    CONST robtarget T4037:=[[56.500013,31.797210,37.750261],[1.000000,0.000000,0.000000,0.000000],[0,0,-1,0],[9E+09,9E+09,9E+09,9E+09,9E+09,9E+09]];
    CONST robtarget T4038:=[[55.000007,31.515698,37.750261],[1.000000,0.000000,0.000000,0.000000],[0,0,-1,0],[9E+09,9E+09,9E+09,9E+09,9E+09,9E+09]];
    CONST robtarget T4039:=[[55.000007,58.695406,37.750261],[1.000000,0.000000,0.000000,0.000000],[0,0,-1,0],[9E+09,9E+09,9E+09,9E+09,9E+09,9E+09]];
    CONST robtarget T4040:=[[53.500001,58.570181,37.750261],[1.000000,0.000000,0.000000,0.000000],[0,0,-1,0],[9E+09,9E+09,9E+09,9E+09,9E+09,9E+09]];
    CONST robtarget T4041:=[[53.500001,31.797216,37.750261],[1.000000,0.000000,0.000000,0.000000],[0,0,-1,0],[9E+09,9E+09,9E+09,9E+09,9E+09,9E+09]];
    CONST robtarget T4042:=[[51.999995,32.435962,37.750261],[1.000000,0.000000,0.000000,0.000000],[0,0,-1,0],[9E+09,9E+09,9E+09,9E+09,9E+09,9E+09]];
    CONST robtarget T4043:=[[51.999995,58.394476,37.750261],[1.000000,0.000000,0.000000,0.000000],[0,0,-1,0],[9E+09,9E+09,9E+09,9E+09,9E+09,9E+09]];
    CONST robtarget T4044:=[[50.499989,57.901720,37.750261],[1.000000,0.000000,0.000000,0.000000],[0,0,-1,0],[9E+09,9E+09,9E+09,9E+09,9E+09,9E+09]];
    CONST robtarget T4045:=[[50.499989,33.195292,37.750261],[1.000000,0.000000,0.000000,0.000000],[0,0,-1,0],[9E+09,9E+09,9E+09,9E+09,9E+09,9E+09]];
    CONST robtarget T4046:=[[48.999983,34.510328,37.750261],[1.000000,0.000000,0.000000,0.000000],[0,0,-1,0],[9E+09,9E+09,9E+09,9E+09,9E+09,9E+09]];
    CONST robtarget T4047:=[[48.999983,57.171733,37.750261],[1.000000,0.000000,0.000000,0.000000],[0,0,-1,0],[9E+09,9E+09,9E+09,9E+09,9E+09,9E+09]];
    CONST robtarget T4048:=[[47.499977,56.303173,37.750261],[1.000000,0.000000,0.000000,0.000000],[0,0,-1,0],[9E+09,9E+09,9E+09,9E+09,9E+09,9E+09]];
    CONST robtarget T4049:=[[47.499977,37.856224,37.750261],[1.000000,0.000000,0.000000,0.000000],[0,0,-1,0],[9E+09,9E+09,9E+09,9E+09,9E+09,9E+09]];
    CONST robtarget T4050:=[[45.999971,39.948571,37.750261],[1.000000,0.000000,0.000000,0.000000],[0,0,-1,0],[9E+09,9E+09,9E+09,9E+09,9E+09,9E+09]];
    CONST robtarget T4051:=[[45.999971,54.916021,37.750261],[1.000000,0.000000,0.000000,0.000000],[0,0,-1,0],[9E+09,9E+09,9E+09,9E+09,9E+09,9E+09]];
    CONST robtarget T4052:=[[44.499965,53.011141,37.750261],[1.000000,0.000000,0.000000,0.000000],[0,0,-1,0],[9E+09,9E+09,9E+09,9E+09,9E+09,9E+09]];
    CONST robtarget T4053:=[[44.499965,42.078797,37.750261],[1.000000,0.000000,0.000000,0.000000],[0,0,-1,0],[9E+09,9E+09,9E+09,9E+09,9E+09,9E+09]];
    CONST robtarget T4054:=[[42.999959,44.372557,37.750261],[1.000000,0.000000,0.000000,0.000000],[0,0,-1,0],[9E+09,9E+09,9E+09,9E+09,9E+09,9E+09]];
    CONST robtarget T4055:=[[42.999959,50.112291,37.750261],[1.000000,0.000000,0.000000,0.000000],[0,0,-1,0],[9E+09,9E+09,9E+09,9E+09,9E+09,9E+09]];
    CONST robtarget T4056:=[[42.999959,44.212149,38.250271],[1.000000,0.000000,0.000000,0.000000],[0,0,-1,0],[9E+09,9E+09,9E+09,9E+09,9E+09,9E+09]];
    CONST robtarget T4057:=[[42.999959,50.185983,38.250271],[1.000000,0.000000,0.000000,0.000000],[0,0,-1,0],[9E+09,9E+09,9E+09,9E+09,9E+09,9E+09]];
    CONST robtarget T4058:=[[42.999959,44.212149,38.250271],[1.000000,0.000000,0.000000,0.000000],[0,0,-1,0],[9E+09,9E+09,9E+09,9E+09,9E+09,9E+09]];
    CONST robtarget T4059:=[[42.999959,50.185983,38.250271],[1.000000,0.000000,0.000000,0.000000],[0,0,-1,0],[9E+09,9E+09,9E+09,9E+09,9E+09,9E+09]];
    CONST robtarget T4060:=[[44.499965,53.123117,38.250271],[1.000000,0.000000,0.000000,0.000000],[0,0,-1,0],[9E+09,9E+09,9E+09,9E+09,9E+09,9E+09]];
    CONST robtarget T4061:=[[44.499965,42.207669,38.250271],[1.000000,0.000000,0.000000,0.000000],[0,0,-1,0],[9E+09,9E+09,9E+09,9E+09,9E+09,9E+09]];
    CONST robtarget T4062:=[[45.999971,40.057127,38.250271],[1.000000,0.000000,0.000000,0.000000],[0,0,-1,0],[9E+09,9E+09,9E+09,9E+09,9E+09,9E+09]];
    CONST robtarget T4063:=[[45.999971,55.075491,38.250271],[1.000000,0.000000,0.000000,0.000000],[0,0,-1,0],[9E+09,9E+09,9E+09,9E+09,9E+09,9E+09]];
    CONST robtarget T4064:=[[47.499977,56.371057,38.250271],[1.000000,0.000000,0.000000,0.000000],[0,0,-1,0],[9E+09,9E+09,9E+09,9E+09,9E+09,9E+09]];
    CONST robtarget T4065:=[[47.499977,38.617217,38.250271],[1.000000,0.000000,0.000000,0.000000],[0,0,-1,0],[9E+09,9E+09,9E+09,9E+09,9E+09,9E+09]];
    CONST robtarget T4066:=[[48.999983,35.664766,38.250271],[1.000000,0.000000,0.000000,0.000000],[0,0,-1,0],[9E+09,9E+09,9E+09,9E+09,9E+09,9E+09]];
    CONST robtarget T4067:=[[48.999983,57.294926,38.250271],[1.000000,0.000000,0.000000,0.000000],[0,0,-1,0],[9E+09,9E+09,9E+09,9E+09,9E+09,9E+09]];
    CONST robtarget T4068:=[[50.499989,58.002093,38.250271],[1.000000,0.000000,0.000000,0.000000],[0,0,-1,0],[9E+09,9E+09,9E+09,9E+09,9E+09,9E+09]];
    CONST robtarget T4069:=[[50.499989,32.700822,38.250271],[1.000000,0.000000,0.000000,0.000000],[0,0,-1,0],[9E+09,9E+09,9E+09,9E+09,9E+09,9E+09]];
    CONST robtarget T4070:=[[51.999995,32.054897,38.250271],[1.000000,0.000000,0.000000,0.000000],[0,0,-1,0],[9E+09,9E+09,9E+09,9E+09,9E+09,9E+09]];
    CONST robtarget T4071:=[[51.999995,58.459231,38.250271],[1.000000,0.000000,0.000000,0.000000],[0,0,-1,0],[9E+09,9E+09,9E+09,9E+09,9E+09,9E+09]];
    CONST robtarget T4072:=[[53.500001,58.647265,38.250271],[1.000000,0.000000,0.000000,0.000000],[0,0,-1,0],[9E+09,9E+09,9E+09,9E+09,9E+09,9E+09]];
    CONST robtarget T4073:=[[53.500001,31.359567,38.250271],[1.000000,0.000000,0.000000,0.000000],[0,0,-1,0],[9E+09,9E+09,9E+09,9E+09,9E+09,9E+09]];
    CONST robtarget T4074:=[[55.000007,31.064300,38.250271],[1.000000,0.000000,0.000000,0.000000],[0,0,-1,0],[9E+09,9E+09,9E+09,9E+09,9E+09,9E+09]];
    CONST robtarget T4075:=[[55.000007,58.772490,38.250271],[1.000000,0.000000,0.000000,0.000000],[0,0,-1,0],[9E+09,9E+09,9E+09,9E+09,9E+09,9E+09]];
    CONST robtarget T4076:=[[56.500013,58.647265,38.250271],[1.000000,0.000000,0.000000,0.000000],[0,0,-1,0],[9E+09,9E+09,9E+09,9E+09,9E+09,9E+09]];
    CONST robtarget T4077:=[[56.500013,31.359567,38.250271],[1.000000,0.000000,0.000000,0.000000],[0,0,-1,0],[9E+09,9E+09,9E+09,9E+09,9E+09,9E+09]];
    CONST robtarget T4078:=[[58.000019,32.054894,38.250271],[1.000000,0.000000,0.000000,0.000000],[0,0,-1,0],[9E+09,9E+09,9E+09,9E+09,9E+09,9E+09]];
    CONST robtarget T4079:=[[58.000019,58.459229,38.250271],[1.000000,0.000000,0.000000,0.000000],[0,0,-1,0],[9E+09,9E+09,9E+09,9E+09,9E+09,9E+09]];
    CONST robtarget T4080:=[[59.500025,58.002093,38.250271],[1.000000,0.000000,0.000000,0.000000],[0,0,-1,0],[9E+09,9E+09,9E+09,9E+09,9E+09,9E+09]];
    CONST robtarget T4081:=[[59.500025,32.700830,38.250271],[1.000000,0.000000,0.000000,0.000000],[0,0,-1,0],[9E+09,9E+09,9E+09,9E+09,9E+09,9E+09]];
    CONST robtarget T4082:=[[61.000031,35.664766,38.250271],[1.000000,0.000000,0.000000,0.000000],[0,0,-1,0],[9E+09,9E+09,9E+09,9E+09,9E+09,9E+09]];
    CONST robtarget T4083:=[[61.000031,57.294925,38.250271],[1.000000,0.000000,0.000000,0.000000],[0,0,-1,0],[9E+09,9E+09,9E+09,9E+09,9E+09,9E+09]];
    CONST robtarget T4084:=[[62.500037,56.371056,38.250271],[1.000000,0.000000,0.000000,0.000000],[0,0,-1,0],[9E+09,9E+09,9E+09,9E+09,9E+09,9E+09]];
    CONST robtarget T4085:=[[62.500037,38.617217,38.250271],[1.000000,0.000000,0.000000,0.000000],[0,0,-1,0],[9E+09,9E+09,9E+09,9E+09,9E+09,9E+09]];
    CONST robtarget T4086:=[[64.000043,40.057127,38.250271],[1.000000,0.000000,0.000000,0.000000],[0,0,-1,0],[9E+09,9E+09,9E+09,9E+09,9E+09,9E+09]];
    CONST robtarget T4087:=[[64.000043,55.075491,38.250271],[1.000000,0.000000,0.000000,0.000000],[0,0,-1,0],[9E+09,9E+09,9E+09,9E+09,9E+09,9E+09]];
    CONST robtarget T4088:=[[65.500049,53.123116,38.250271],[1.000000,0.000000,0.000000,0.000000],[0,0,-1,0],[9E+09,9E+09,9E+09,9E+09,9E+09,9E+09]];
    CONST robtarget T4089:=[[65.500049,42.207669,38.250271],[1.000000,0.000000,0.000000,0.000000],[0,0,-1,0],[9E+09,9E+09,9E+09,9E+09,9E+09,9E+09]];
    CONST robtarget T4090:=[[67.000055,44.212149,38.250271],[1.000000,0.000000,0.000000,0.000000],[0,0,-1,0],[9E+09,9E+09,9E+09,9E+09,9E+09,9E+09]];
    CONST robtarget T4091:=[[67.000055,50.185984,38.250271],[1.000000,0.000000,0.000000,0.000000],[0,0,-1,0],[9E+09,9E+09,9E+09,9E+09,9E+09,9E+09]];
    CONST robtarget T4092:=[[67.000055,44.131949,38.750281],[1.000000,0.000000,0.000000,0.000000],[0,0,-1,0],[9E+09,9E+09,9E+09,9E+09,9E+09,9E+09]];
    CONST robtarget T4093:=[[67.000055,50.259676,38.750281],[1.000000,0.000000,0.000000,0.000000],[0,0,-1,0],[9E+09,9E+09,9E+09,9E+09,9E+09,9E+09]];
    CONST robtarget T4094:=[[67.000055,44.131949,38.750281],[1.000000,0.000000,0.000000,0.000000],[0,0,-1,0],[9E+09,9E+09,9E+09,9E+09,9E+09,9E+09]];
    CONST robtarget T4095:=[[67.000055,50.259676,38.750281],[1.000000,0.000000,0.000000,0.000000],[0,0,-1,0],[9E+09,9E+09,9E+09,9E+09,9E+09,9E+09]];
    CONST robtarget T4096:=[[65.500049,53.235088,38.750281],[1.000000,0.000000,0.000000,0.000000],[0,0,-1,0],[9E+09,9E+09,9E+09,9E+09,9E+09,9E+09]];
    CONST robtarget T4097:=[[65.500049,42.336541,38.750281],[1.000000,0.000000,0.000000,0.000000],[0,0,-1,0],[9E+09,9E+09,9E+09,9E+09,9E+09,9E+09]];
    CONST robtarget T4098:=[[64.000043,40.167265,38.750281],[1.000000,0.000000,0.000000,0.000000],[0,0,-1,0],[9E+09,9E+09,9E+09,9E+09,9E+09,9E+09]];
    CONST robtarget T4099:=[[64.000043,55.123261,38.750281],[1.000000,0.000000,0.000000,0.000000],[0,0,-1,0],[9E+09,9E+09,9E+09,9E+09,9E+09,9E+09]];
    CONST robtarget T4100:=[[62.500037,56.438940,38.750281],[1.000000,0.000000,0.000000,0.000000],[0,0,-1,0],[9E+09,9E+09,9E+09,9E+09,9E+09,9E+09]];
    CONST robtarget T4101:=[[62.500037,38.816896,38.750281],[1.000000,0.000000,0.000000,0.000000],[0,0,-1,0],[9E+09,9E+09,9E+09,9E+09,9E+09,9E+09]];
    CONST robtarget T4102:=[[61.000031,36.698545,38.750281],[1.000000,0.000000,0.000000,0.000000],[0,0,-1,0],[9E+09,9E+09,9E+09,9E+09,9E+09,9E+09]];
    CONST robtarget T4103:=[[61.000031,57.398916,38.750281],[1.000000,0.000000,0.000000,0.000000],[0,0,-1,0],[9E+09,9E+09,9E+09,9E+09,9E+09,9E+09]];
    CONST robtarget T4104:=[[59.500025,58.045436,38.750281],[1.000000,0.000000,0.000000,0.000000],[0,0,-1,0],[9E+09,9E+09,9E+09,9E+09,9E+09,9E+09]];
    CONST robtarget T4105:=[[59.500025,32.999058,38.750281],[1.000000,0.000000,0.000000,0.000000],[0,0,-1,0],[9E+09,9E+09,9E+09,9E+09,9E+09,9E+09]];
    CONST robtarget T4106:=[[58.000019,31.695724,38.750281],[1.000000,0.000000,0.000000,0.000000],[0,0,-1,0],[9E+09,9E+09,9E+09,9E+09,9E+09,9E+09]];
    CONST robtarget T4107:=[[58.000019,58.532197,38.750281],[1.000000,0.000000,0.000000,0.000000],[0,0,-1,0],[9E+09,9E+09,9E+09,9E+09,9E+09,9E+09]];
    CONST robtarget T4108:=[[56.500013,58.721504,38.750281],[1.000000,0.000000,0.000000,0.000000],[0,0,-1,0],[9E+09,9E+09,9E+09,9E+09,9E+09,9E+09]];
    CONST robtarget T4109:=[[56.500013,30.999539,38.750281],[1.000000,0.000000,0.000000,0.000000],[0,0,-1,0],[9E+09,9E+09,9E+09,9E+09,9E+09,9E+09]];
    CONST robtarget T4110:=[[55.000007,30.672510,38.750281],[1.000000,0.000000,0.000000,0.000000],[0,0,-1,0],[9E+09,9E+09,9E+09,9E+09,9E+09,9E+09]];
    CONST robtarget T4111:=[[55.000007,58.849574,38.750281],[1.000000,0.000000,0.000000,0.000000],[0,0,-1,0],[9E+09,9E+09,9E+09,9E+09,9E+09,9E+09]];
    CONST robtarget T4112:=[[53.500001,58.721507,38.750281],[1.000000,0.000000,0.000000,0.000000],[0,0,-1,0],[9E+09,9E+09,9E+09,9E+09,9E+09,9E+09]];
    CONST robtarget T4113:=[[53.500001,30.999539,38.750281],[1.000000,0.000000,0.000000,0.000000],[0,0,-1,0],[9E+09,9E+09,9E+09,9E+09,9E+09,9E+09]];
    CONST robtarget T4114:=[[51.999995,31.695723,38.750281],[1.000000,0.000000,0.000000,0.000000],[0,0,-1,0],[9E+09,9E+09,9E+09,9E+09,9E+09,9E+09]];
    CONST robtarget T4115:=[[51.999995,58.532203,38.750281],[1.000000,0.000000,0.000000,0.000000],[0,0,-1,0],[9E+09,9E+09,9E+09,9E+09,9E+09,9E+09]];
    CONST robtarget T4116:=[[50.499989,58.045436,38.750281],[1.000000,0.000000,0.000000,0.000000],[0,0,-1,0],[9E+09,9E+09,9E+09,9E+09,9E+09,9E+09]];
    CONST robtarget T4117:=[[50.499989,32.999059,38.750281],[1.000000,0.000000,0.000000,0.000000],[0,0,-1,0],[9E+09,9E+09,9E+09,9E+09,9E+09,9E+09]];
    CONST robtarget T4118:=[[48.999983,36.698544,38.750281],[1.000000,0.000000,0.000000,0.000000],[0,0,-1,0],[9E+09,9E+09,9E+09,9E+09,9E+09,9E+09]];
    CONST robtarget T4119:=[[48.999983,57.398916,38.750281],[1.000000,0.000000,0.000000,0.000000],[0,0,-1,0],[9E+09,9E+09,9E+09,9E+09,9E+09,9E+09]];
    CONST robtarget T4120:=[[47.499977,56.438941,38.750281],[1.000000,0.000000,0.000000,0.000000],[0,0,-1,0],[9E+09,9E+09,9E+09,9E+09,9E+09,9E+09]];
    CONST robtarget T4121:=[[47.499977,38.816896,38.750281],[1.000000,0.000000,0.000000,0.000000],[0,0,-1,0],[9E+09,9E+09,9E+09,9E+09,9E+09,9E+09]];
    CONST robtarget T4122:=[[45.999971,40.167264,38.750281],[1.000000,0.000000,0.000000,0.000000],[0,0,-1,0],[9E+09,9E+09,9E+09,9E+09,9E+09,9E+09]];
    CONST robtarget T4123:=[[45.999971,55.123261,38.750281],[1.000000,0.000000,0.000000,0.000000],[0,0,-1,0],[9E+09,9E+09,9E+09,9E+09,9E+09,9E+09]];
    CONST robtarget T4124:=[[44.499965,53.235093,38.750281],[1.000000,0.000000,0.000000,0.000000],[0,0,-1,0],[9E+09,9E+09,9E+09,9E+09,9E+09,9E+09]];
    CONST robtarget T4125:=[[44.499965,42.336540,38.750281],[1.000000,0.000000,0.000000,0.000000],[0,0,-1,0],[9E+09,9E+09,9E+09,9E+09,9E+09,9E+09]];
    CONST robtarget T4126:=[[42.999959,44.131948,38.750281],[1.000000,0.000000,0.000000,0.000000],[0,0,-1,0],[9E+09,9E+09,9E+09,9E+09,9E+09,9E+09]];
    CONST robtarget T4127:=[[42.999959,50.259676,38.750281],[1.000000,0.000000,0.000000,0.000000],[0,0,-1,0],[9E+09,9E+09,9E+09,9E+09,9E+09,9E+09]];
    CONST robtarget T4128:=[[42.999959,44.054116,39.250291],[1.000000,0.000000,0.000000,0.000000],[0,0,-1,0],[9E+09,9E+09,9E+09,9E+09,9E+09,9E+09]];
    CONST robtarget T4129:=[[42.999959,50.376289,39.250291],[1.000000,0.000000,0.000000,0.000000],[0,0,-1,0],[9E+09,9E+09,9E+09,9E+09,9E+09,9E+09]];
    CONST robtarget T4130:=[[42.999959,44.054116,39.250291],[1.000000,0.000000,0.000000,0.000000],[0,0,-1,0],[9E+09,9E+09,9E+09,9E+09,9E+09,9E+09]];
    CONST robtarget T4131:=[[42.999959,50.376289,39.250291],[1.000000,0.000000,0.000000,0.000000],[0,0,-1,0],[9E+09,9E+09,9E+09,9E+09,9E+09,9E+09]];
    CONST robtarget T4132:=[[44.499965,53.135053,39.250291],[1.000000,0.000000,0.000000,0.000000],[0,0,-1,0],[9E+09,9E+09,9E+09,9E+09,9E+09,9E+09]];
    CONST robtarget T4133:=[[44.499965,42.332431,39.250291],[1.000000,0.000000,0.000000,0.000000],[0,0,-1,0],[9E+09,9E+09,9E+09,9E+09,9E+09,9E+09]];
    CONST robtarget T4134:=[[45.999971,40.374790,39.250291],[1.000000,0.000000,0.000000,0.000000],[0,0,-1,0],[9E+09,9E+09,9E+09,9E+09,9E+09,9E+09]];
    CONST robtarget T4135:=[[45.999971,55.113414,39.250291],[1.000000,0.000000,0.000000,0.000000],[0,0,-1,0],[9E+09,9E+09,9E+09,9E+09,9E+09,9E+09]];
    CONST robtarget T4136:=[[47.499977,56.506825,39.250291],[1.000000,0.000000,0.000000,0.000000],[0,0,-1,0],[9E+09,9E+09,9E+09,9E+09,9E+09,9E+09]];
    CONST robtarget T4137:=[[47.499977,38.996522,39.250291],[1.000000,0.000000,0.000000,0.000000],[0,0,-1,0],[9E+09,9E+09,9E+09,9E+09,9E+09,9E+09]];
    CONST robtarget T4138:=[[48.999983,37.580618,39.250291],[1.000000,0.000000,0.000000,0.000000],[0,0,-1,0],[9E+09,9E+09,9E+09,9E+09,9E+09,9E+09]];
    CONST robtarget T4139:=[[48.999983,57.420832,39.250291],[1.000000,0.000000,0.000000,0.000000],[0,0,-1,0],[9E+09,9E+09,9E+09,9E+09,9E+09,9E+09]];
    CONST robtarget T4140:=[[50.499989,58.088778,39.250291],[1.000000,0.000000,0.000000,0.000000],[0,0,-1,0],[9E+09,9E+09,9E+09,9E+09,9E+09,9E+09]];
    CONST robtarget T4141:=[[50.499989,34.138448,39.250291],[1.000000,0.000000,0.000000,0.000000],[0,0,-1,0],[9E+09,9E+09,9E+09,9E+09,9E+09,9E+09]];
    CONST robtarget T4142:=[[51.999995,31.384926,39.250291],[1.000000,0.000000,0.000000,0.000000],[0,0,-1,0],[9E+09,9E+09,9E+09,9E+09,9E+09,9E+09]];
    CONST robtarget T4143:=[[51.999995,58.605174,39.250291],[1.000000,0.000000,0.000000,0.000000],[0,0,-1,0],[9E+09,9E+09,9E+09,9E+09,9E+09,9E+09]];
    CONST robtarget T4144:=[[53.500001,58.780455,39.250291],[1.000000,0.000000,0.000000,0.000000],[0,0,-1,0],[9E+09,9E+09,9E+09,9E+09,9E+09,9E+09]];
    CONST robtarget T4145:=[[53.500001,30.721918,39.250291],[1.000000,0.000000,0.000000,0.000000],[0,0,-1,0],[9E+09,9E+09,9E+09,9E+09,9E+09,9E+09]];
    CONST robtarget T4146:=[[55.000007,30.347257,39.250291],[1.000000,0.000000,0.000000,0.000000],[0,0,-1,0],[9E+09,9E+09,9E+09,9E+09,9E+09,9E+09]];
    CONST robtarget T4147:=[[55.000007,58.890261,39.250291],[1.000000,0.000000,0.000000,0.000000],[0,0,-1,0],[9E+09,9E+09,9E+09,9E+09,9E+09,9E+09]];
    CONST robtarget T4148:=[[56.500013,58.780450,39.250291],[1.000000,0.000000,0.000000,0.000000],[0,0,-1,0],[9E+09,9E+09,9E+09,9E+09,9E+09,9E+09]];
    CONST robtarget T4149:=[[56.500013,30.721922,39.250291],[1.000000,0.000000,0.000000,0.000000],[0,0,-1,0],[9E+09,9E+09,9E+09,9E+09,9E+09,9E+09]];
    CONST robtarget T4150:=[[58.000019,31.384926,39.250291],[1.000000,0.000000,0.000000,0.000000],[0,0,-1,0],[9E+09,9E+09,9E+09,9E+09,9E+09,9E+09]];
    CONST robtarget T4151:=[[58.000019,58.605166,39.250291],[1.000000,0.000000,0.000000,0.000000],[0,0,-1,0],[9E+09,9E+09,9E+09,9E+09,9E+09,9E+09]];
    CONST robtarget T4152:=[[59.500025,58.088778,39.250291],[1.000000,0.000000,0.000000,0.000000],[0,0,-1,0],[9E+09,9E+09,9E+09,9E+09,9E+09,9E+09]];
    CONST robtarget T4153:=[[59.500025,34.138448,39.250291],[1.000000,0.000000,0.000000,0.000000],[0,0,-1,0],[9E+09,9E+09,9E+09,9E+09,9E+09,9E+09]];
    CONST robtarget T4154:=[[61.000031,37.580618,39.250291],[1.000000,0.000000,0.000000,0.000000],[0,0,-1,0],[9E+09,9E+09,9E+09,9E+09,9E+09,9E+09]];
    CONST robtarget T4155:=[[61.000031,57.420832,39.250291],[1.000000,0.000000,0.000000,0.000000],[0,0,-1,0],[9E+09,9E+09,9E+09,9E+09,9E+09,9E+09]];
    CONST robtarget T4156:=[[62.500037,56.506824,39.250291],[1.000000,0.000000,0.000000,0.000000],[0,0,-1,0],[9E+09,9E+09,9E+09,9E+09,9E+09,9E+09]];
    CONST robtarget T4157:=[[62.500037,38.996523,39.250291],[1.000000,0.000000,0.000000,0.000000],[0,0,-1,0],[9E+09,9E+09,9E+09,9E+09,9E+09,9E+09]];
    CONST robtarget T4158:=[[64.000043,40.374792,39.250291],[1.000000,0.000000,0.000000,0.000000],[0,0,-1,0],[9E+09,9E+09,9E+09,9E+09,9E+09,9E+09]];
    CONST robtarget T4159:=[[64.000043,55.113414,39.250291],[1.000000,0.000000,0.000000,0.000000],[0,0,-1,0],[9E+09,9E+09,9E+09,9E+09,9E+09,9E+09]];
    CONST robtarget T4160:=[[65.500049,53.135049,39.250291],[1.000000,0.000000,0.000000,0.000000],[0,0,-1,0],[9E+09,9E+09,9E+09,9E+09,9E+09,9E+09]];
    CONST robtarget T4161:=[[65.500049,42.332431,39.250291],[1.000000,0.000000,0.000000,0.000000],[0,0,-1,0],[9E+09,9E+09,9E+09,9E+09,9E+09,9E+09]];
    CONST robtarget T4162:=[[67.000055,44.054117,39.250291],[1.000000,0.000000,0.000000,0.000000],[0,0,-1,0],[9E+09,9E+09,9E+09,9E+09,9E+09,9E+09]];
    CONST robtarget T4163:=[[67.000055,50.376286,39.250291],[1.000000,0.000000,0.000000,0.000000],[0,0,-1,0],[9E+09,9E+09,9E+09,9E+09,9E+09,9E+09]];
    CONST robtarget T4164:=[[67.000055,44.072887,39.750301],[1.000000,0.000000,0.000000,0.000000],[0,0,-1,0],[9E+09,9E+09,9E+09,9E+09,9E+09,9E+09]];
    CONST robtarget T4165:=[[67.000055,50.303617,39.750301],[1.000000,0.000000,0.000000,0.000000],[0,0,-1,0],[9E+09,9E+09,9E+09,9E+09,9E+09,9E+09]];
    CONST robtarget T4166:=[[67.000055,44.072887,39.750301],[1.000000,0.000000,0.000000,0.000000],[0,0,-1,0],[9E+09,9E+09,9E+09,9E+09,9E+09,9E+09]];
    CONST robtarget T4167:=[[67.000055,50.303617,39.750301],[1.000000,0.000000,0.000000,0.000000],[0,0,-1,0],[9E+09,9E+09,9E+09,9E+09,9E+09,9E+09]];
    CONST robtarget T4168:=[[65.500049,52.995505,39.750301],[1.000000,0.000000,0.000000,0.000000],[0,0,-1,0],[9E+09,9E+09,9E+09,9E+09,9E+09,9E+09]];
    CONST robtarget T4169:=[[65.500049,42.422914,39.750301],[1.000000,0.000000,0.000000,0.000000],[0,0,-1,0],[9E+09,9E+09,9E+09,9E+09,9E+09,9E+09]];
    CONST robtarget T4170:=[[64.000043,40.653208,39.750301],[1.000000,0.000000,0.000000,0.000000],[0,0,-1,0],[9E+09,9E+09,9E+09,9E+09,9E+09,9E+09]];
    CONST robtarget T4171:=[[64.000043,55.084923,39.750301],[1.000000,0.000000,0.000000,0.000000],[0,0,-1,0],[9E+09,9E+09,9E+09,9E+09,9E+09,9E+09]];
    CONST robtarget T4172:=[[62.500037,56.521256,39.750301],[1.000000,0.000000,0.000000,0.000000],[0,0,-1,0],[9E+09,9E+09,9E+09,9E+09,9E+09,9E+09]];
    CONST robtarget T4173:=[[62.500037,39.193232,39.750301],[1.000000,0.000000,0.000000,0.000000],[0,0,-1,0],[9E+09,9E+09,9E+09,9E+09,9E+09,9E+09]];
    CONST robtarget T4174:=[[61.000031,38.058259,39.750301],[1.000000,0.000000,0.000000,0.000000],[0,0,-1,0],[9E+09,9E+09,9E+09,9E+09,9E+09,9E+09]];
    CONST robtarget T4175:=[[61.000031,57.442748,39.750301],[1.000000,0.000000,0.000000,0.000000],[0,0,-1,0],[9E+09,9E+09,9E+09,9E+09,9E+09,9E+09]];
    CONST robtarget T4176:=[[59.500025,58.151010,39.750301],[1.000000,0.000000,0.000000,0.000000],[0,0,-1,0],[9E+09,9E+09,9E+09,9E+09,9E+09,9E+09]];
    CONST robtarget T4177:=[[59.500025,35.190368,39.750301],[1.000000,0.000000,0.000000,0.000000],[0,0,-1,0],[9E+09,9E+09,9E+09,9E+09,9E+09,9E+09]];
    CONST robtarget T4178:=[[58.000019,31.632069,39.750301],[1.000000,0.000000,0.000000,0.000000],[0,0,-1,0],[9E+09,9E+09,9E+09,9E+09,9E+09,9E+09]];
    CONST robtarget T4179:=[[58.000019,58.594733,39.750301],[1.000000,0.000000,0.000000,0.000000],[0,0,-1,0],[9E+09,9E+09,9E+09,9E+09,9E+09,9E+09]];
    CONST robtarget T4180:=[[56.500013,58.779478,39.750301],[1.000000,0.000000,0.000000,0.000000],[0,0,-1,0],[9E+09,9E+09,9E+09,9E+09,9E+09,9E+09]];
    CONST robtarget T4181:=[[56.500013,30.692136,39.750301],[1.000000,0.000000,0.000000,0.000000],[0,0,-1,0],[9E+09,9E+09,9E+09,9E+09,9E+09,9E+09]];
    CONST robtarget T4182:=[[55.000007,30.109747,39.750301],[1.000000,0.000000,0.000000,0.000000],[0,0,-1,0],[9E+09,9E+09,9E+09,9E+09,9E+09,9E+09]];
    CONST robtarget T4183:=[[55.000007,58.885895,39.750301],[1.000000,0.000000,0.000000,0.000000],[0,0,-1,0],[9E+09,9E+09,9E+09,9E+09,9E+09,9E+09]];
    CONST robtarget T4184:=[[53.500001,58.779480,39.750301],[1.000000,0.000000,0.000000,0.000000],[0,0,-1,0],[9E+09,9E+09,9E+09,9E+09,9E+09,9E+09]];
    CONST robtarget T4185:=[[53.500001,30.692135,39.750301],[1.000000,0.000000,0.000000,0.000000],[0,0,-1,0],[9E+09,9E+09,9E+09,9E+09,9E+09,9E+09]];
    CONST robtarget T4186:=[[51.999995,31.632069,39.750301],[1.000000,0.000000,0.000000,0.000000],[0,0,-1,0],[9E+09,9E+09,9E+09,9E+09,9E+09,9E+09]];
    CONST robtarget T4187:=[[51.999995,58.594739,39.750301],[1.000000,0.000000,0.000000,0.000000],[0,0,-1,0],[9E+09,9E+09,9E+09,9E+09,9E+09,9E+09]];
    CONST robtarget T4188:=[[50.499989,58.151012,39.750301],[1.000000,0.000000,0.000000,0.000000],[0,0,-1,0],[9E+09,9E+09,9E+09,9E+09,9E+09,9E+09]];
    CONST robtarget T4189:=[[50.499989,35.190377,39.750301],[1.000000,0.000000,0.000000,0.000000],[0,0,-1,0],[9E+09,9E+09,9E+09,9E+09,9E+09,9E+09]];
    CONST robtarget T4190:=[[48.999983,38.058258,39.750301],[1.000000,0.000000,0.000000,0.000000],[0,0,-1,0],[9E+09,9E+09,9E+09,9E+09,9E+09,9E+09]];
    CONST robtarget T4191:=[[48.999983,57.442748,39.750301],[1.000000,0.000000,0.000000,0.000000],[0,0,-1,0],[9E+09,9E+09,9E+09,9E+09,9E+09,9E+09]];
    CONST robtarget T4192:=[[47.499977,56.521257,39.750301],[1.000000,0.000000,0.000000,0.000000],[0,0,-1,0],[9E+09,9E+09,9E+09,9E+09,9E+09,9E+09]];
    CONST robtarget T4193:=[[47.499977,39.193232,39.750301],[1.000000,0.000000,0.000000,0.000000],[0,0,-1,0],[9E+09,9E+09,9E+09,9E+09,9E+09,9E+09]];
    CONST robtarget T4194:=[[45.999971,40.653206,39.750301],[1.000000,0.000000,0.000000,0.000000],[0,0,-1,0],[9E+09,9E+09,9E+09,9E+09,9E+09,9E+09]];
    CONST robtarget T4195:=[[45.999971,55.084923,39.750301],[1.000000,0.000000,0.000000,0.000000],[0,0,-1,0],[9E+09,9E+09,9E+09,9E+09,9E+09,9E+09]];
    CONST robtarget T4196:=[[44.499965,52.995507,39.750301],[1.000000,0.000000,0.000000,0.000000],[0,0,-1,0],[9E+09,9E+09,9E+09,9E+09,9E+09,9E+09]];
    CONST robtarget T4197:=[[44.499965,42.422914,39.750301],[1.000000,0.000000,0.000000,0.000000],[0,0,-1,0],[9E+09,9E+09,9E+09,9E+09,9E+09,9E+09]];
    CONST robtarget T4198:=[[42.999959,44.072887,39.750301],[1.000000,0.000000,0.000000,0.000000],[0,0,-1,0],[9E+09,9E+09,9E+09,9E+09,9E+09,9E+09]];
    CONST robtarget T4199:=[[42.999959,50.303618,39.750301],[1.000000,0.000000,0.000000,0.000000],[0,0,-1,0],[9E+09,9E+09,9E+09,9E+09,9E+09,9E+09]];
    CONST robtarget T4200:=[[42.999959,43.957416,40.250311],[1.000000,0.000000,0.000000,0.000000],[0,0,-1,0],[9E+09,9E+09,9E+09,9E+09,9E+09,9E+09]];
    CONST robtarget T4201:=[[42.999959,50.041103,40.250311],[1.000000,0.000000,0.000000,0.000000],[0,0,-1,0],[9E+09,9E+09,9E+09,9E+09,9E+09,9E+09]];
    CONST robtarget T4202:=[[42.999959,43.957416,40.250311],[1.000000,0.000000,0.000000,0.000000],[0,0,-1,0],[9E+09,9E+09,9E+09,9E+09,9E+09,9E+09]];
    CONST robtarget T4203:=[[42.999959,50.041103,40.250311],[1.000000,0.000000,0.000000,0.000000],[0,0,-1,0],[9E+09,9E+09,9E+09,9E+09,9E+09,9E+09]];
    CONST robtarget T4204:=[[44.499965,52.855961,40.250311],[1.000000,0.000000,0.000000,0.000000],[0,0,-1,0],[9E+09,9E+09,9E+09,9E+09,9E+09,9E+09]];
    CONST robtarget T4205:=[[44.499965,42.549901,40.250311],[1.000000,0.000000,0.000000,0.000000],[0,0,-1,0],[9E+09,9E+09,9E+09,9E+09,9E+09,9E+09]];
    CONST robtarget T4206:=[[45.999971,40.933620,40.250311],[1.000000,0.000000,0.000000,0.000000],[0,0,-1,0],[9E+09,9E+09,9E+09,9E+09,9E+09,9E+09]];
    CONST robtarget T4207:=[[45.999971,55.056432,40.250311],[1.000000,0.000000,0.000000,0.000000],[0,0,-1,0],[9E+09,9E+09,9E+09,9E+09,9E+09,9E+09]];
    CONST robtarget T4208:=[[47.499977,56.418593,40.250311],[1.000000,0.000000,0.000000,0.000000],[0,0,-1,0],[9E+09,9E+09,9E+09,9E+09,9E+09,9E+09]];
    CONST robtarget T4209:=[[47.499977,39.361755,40.250311],[1.000000,0.000000,0.000000,0.000000],[0,0,-1,0],[9E+09,9E+09,9E+09,9E+09,9E+09,9E+09]];
    CONST robtarget T4210:=[[48.999983,38.258018,40.250311],[1.000000,0.000000,0.000000,0.000000],[0,0,-1,0],[9E+09,9E+09,9E+09,9E+09,9E+09,9E+09]];
    CONST robtarget T4211:=[[48.999983,57.406745,40.250311],[1.000000,0.000000,0.000000,0.000000],[0,0,-1,0],[9E+09,9E+09,9E+09,9E+09,9E+09,9E+09]];
    CONST robtarget T4212:=[[50.499989,58.142889,40.250311],[1.000000,0.000000,0.000000,0.000000],[0,0,-1,0],[9E+09,9E+09,9E+09,9E+09,9E+09,9E+09]];
    CONST robtarget T4213:=[[50.499989,36.203320,40.250311],[1.000000,0.000000,0.000000,0.000000],[0,0,-1,0],[9E+09,9E+09,9E+09,9E+09,9E+09,9E+09]];
    CONST robtarget T4214:=[[51.999995,32.225362,40.250311],[1.000000,0.000000,0.000000,0.000000],[0,0,-1,0],[9E+09,9E+09,9E+09,9E+09,9E+09,9E+09]];
    CONST robtarget T4215:=[[51.999995,58.567705,40.250311],[1.000000,0.000000,0.000000,0.000000],[0,0,-1,0],[9E+09,9E+09,9E+09,9E+09,9E+09,9E+09]];
    CONST robtarget T4216:=[[53.500001,58.777623,40.250311],[1.000000,0.000000,0.000000,0.000000],[0,0,-1,0],[9E+09,9E+09,9E+09,9E+09,9E+09,9E+09]];
    CONST robtarget T4217:=[[53.500001,30.491220,40.250311],[1.000000,0.000000,0.000000,0.000000],[0,0,-1,0],[9E+09,9E+09,9E+09,9E+09,9E+09,9E+09]];
    CONST robtarget T4218:=[[55.000007,30.188626,40.250311],[1.000000,0.000000,0.000000,0.000000],[0,0,-1,0],[9E+09,9E+09,9E+09,9E+09,9E+09,9E+09]];
    CONST robtarget T4219:=[[55.000007,58.881529,40.250311],[1.000000,0.000000,0.000000,0.000000],[0,0,-1,0],[9E+09,9E+09,9E+09,9E+09,9E+09,9E+09]];
    CONST robtarget T4220:=[[56.500013,58.777623,40.250311],[1.000000,0.000000,0.000000,0.000000],[0,0,-1,0],[9E+09,9E+09,9E+09,9E+09,9E+09,9E+09]];
    CONST robtarget T4221:=[[56.500013,30.491221,40.250311],[1.000000,0.000000,0.000000,0.000000],[0,0,-1,0],[9E+09,9E+09,9E+09,9E+09,9E+09,9E+09]];
    CONST robtarget T4222:=[[58.000019,32.225362,40.250311],[1.000000,0.000000,0.000000,0.000000],[0,0,-1,0],[9E+09,9E+09,9E+09,9E+09,9E+09,9E+09]];
    CONST robtarget T4223:=[[58.000019,58.567702,40.250311],[1.000000,0.000000,0.000000,0.000000],[0,0,-1,0],[9E+09,9E+09,9E+09,9E+09,9E+09,9E+09]];
    CONST robtarget T4224:=[[59.500025,58.142889,40.250311],[1.000000,0.000000,0.000000,0.000000],[0,0,-1,0],[9E+09,9E+09,9E+09,9E+09,9E+09,9E+09]];
    CONST robtarget T4225:=[[59.500025,36.203317,40.250311],[1.000000,0.000000,0.000000,0.000000],[0,0,-1,0],[9E+09,9E+09,9E+09,9E+09,9E+09,9E+09]];
    CONST robtarget T4226:=[[61.000031,38.258019,40.250311],[1.000000,0.000000,0.000000,0.000000],[0,0,-1,0],[9E+09,9E+09,9E+09,9E+09,9E+09,9E+09]];
    CONST robtarget T4227:=[[61.000031,57.406746,40.250311],[1.000000,0.000000,0.000000,0.000000],[0,0,-1,0],[9E+09,9E+09,9E+09,9E+09,9E+09,9E+09]];
    CONST robtarget T4228:=[[62.500037,56.418593,40.250311],[1.000000,0.000000,0.000000,0.000000],[0,0,-1,0],[9E+09,9E+09,9E+09,9E+09,9E+09,9E+09]];
    CONST robtarget T4229:=[[62.500037,39.361755,40.250311],[1.000000,0.000000,0.000000,0.000000],[0,0,-1,0],[9E+09,9E+09,9E+09,9E+09,9E+09,9E+09]];
    CONST robtarget T4230:=[[64.000043,40.933621,40.250311],[1.000000,0.000000,0.000000,0.000000],[0,0,-1,0],[9E+09,9E+09,9E+09,9E+09,9E+09,9E+09]];
    CONST robtarget T4231:=[[64.000043,55.056432,40.250311],[1.000000,0.000000,0.000000,0.000000],[0,0,-1,0],[9E+09,9E+09,9E+09,9E+09,9E+09,9E+09]];
    CONST robtarget T4232:=[[65.500049,52.855961,40.250311],[1.000000,0.000000,0.000000,0.000000],[0,0,-1,0],[9E+09,9E+09,9E+09,9E+09,9E+09,9E+09]];
    CONST robtarget T4233:=[[65.500049,42.549900,40.250311],[1.000000,0.000000,0.000000,0.000000],[0,0,-1,0],[9E+09,9E+09,9E+09,9E+09,9E+09,9E+09]];
    CONST robtarget T4234:=[[67.000055,43.957416,40.250311],[1.000000,0.000000,0.000000,0.000000],[0,0,-1,0],[9E+09,9E+09,9E+09,9E+09,9E+09,9E+09]];
    CONST robtarget T4235:=[[67.000055,50.041104,40.250311],[1.000000,0.000000,0.000000,0.000000],[0,0,-1,0],[9E+09,9E+09,9E+09,9E+09,9E+09,9E+09]];
    CONST robtarget T4236:=[[67.000060,43.826036,40.750321],[1.000000,0.000000,0.000000,0.000000],[0,0,-1,0],[9E+09,9E+09,9E+09,9E+09,9E+09,9E+09]];
    CONST robtarget T4237:=[[67.000060,49.731609,40.750321],[1.000000,0.000000,0.000000,0.000000],[0,0,-1,0],[9E+09,9E+09,9E+09,9E+09,9E+09,9E+09]];
    CONST robtarget T4238:=[[67.000060,43.826036,40.750321],[1.000000,0.000000,0.000000,0.000000],[0,0,-1,0],[9E+09,9E+09,9E+09,9E+09,9E+09,9E+09]];
    CONST robtarget T4239:=[[67.000060,49.731609,40.750321],[1.000000,0.000000,0.000000,0.000000],[0,0,-1,0],[9E+09,9E+09,9E+09,9E+09,9E+09,9E+09]];
    CONST robtarget T4240:=[[65.500054,52.723909,40.750321],[1.000000,0.000000,0.000000,0.000000],[0,0,-1,0],[9E+09,9E+09,9E+09,9E+09,9E+09,9E+09]];
    CONST robtarget T4241:=[[65.500054,42.646321,40.750321],[1.000000,0.000000,0.000000,0.000000],[0,0,-1,0],[9E+09,9E+09,9E+09,9E+09,9E+09,9E+09]];
    CONST robtarget T4242:=[[64.000048,41.154252,40.750321],[1.000000,0.000000,0.000000,0.000000],[0,0,-1,0],[9E+09,9E+09,9E+09,9E+09,9E+09,9E+09]];
    CONST robtarget T4243:=[[64.000048,54.938664,40.750321],[1.000000,0.000000,0.000000,0.000000],[0,0,-1,0],[9E+09,9E+09,9E+09,9E+09,9E+09,9E+09]];
    CONST robtarget T4244:=[[62.500042,56.300294,40.750321],[1.000000,0.000000,0.000000,0.000000],[0,0,-1,0],[9E+09,9E+09,9E+09,9E+09,9E+09,9E+09]];
    CONST robtarget T4245:=[[62.500042,39.555182,40.750321],[1.000000,0.000000,0.000000,0.000000],[0,0,-1,0],[9E+09,9E+09,9E+09,9E+09,9E+09,9E+09]];
    CONST robtarget T4246:=[[61.000036,38.408170,40.750321],[1.000000,0.000000,0.000000,0.000000],[0,0,-1,0],[9E+09,9E+09,9E+09,9E+09,9E+09,9E+09]];
    CONST robtarget T4247:=[[61.000036,57.345134,40.750321],[1.000000,0.000000,0.000000,0.000000],[0,0,-1,0],[9E+09,9E+09,9E+09,9E+09,9E+09,9E+09]];
    CONST robtarget T4248:=[[59.500030,58.096457,40.750321],[1.000000,0.000000,0.000000,0.000000],[0,0,-1,0],[9E+09,9E+09,9E+09,9E+09,9E+09,9E+09]];
    CONST robtarget T4249:=[[59.500030,37.166192,40.750321],[1.000000,0.000000,0.000000,0.000000],[0,0,-1,0],[9E+09,9E+09,9E+09,9E+09,9E+09,9E+09]];
    CONST robtarget T4250:=[[58.000024,33.123119,40.750321],[1.000000,0.000000,0.000000,0.000000],[0,0,-1,0],[9E+09,9E+09,9E+09,9E+09,9E+09,9E+09]];
    CONST robtarget T4251:=[[58.000024,58.535315,40.750321],[1.000000,0.000000,0.000000,0.000000],[0,0,-1,0],[9E+09,9E+09,9E+09,9E+09,9E+09,9E+09]];
    CONST robtarget T4252:=[[56.500018,58.762255,40.750321],[1.000000,0.000000,0.000000,0.000000],[0,0,-1,0],[9E+09,9E+09,9E+09,9E+09,9E+09,9E+09]];
    CONST robtarget T4253:=[[56.500018,30.483209,40.750321],[1.000000,0.000000,0.000000,0.000000],[0,0,-1,0],[9E+09,9E+09,9E+09,9E+09,9E+09,9E+09]];
    CONST robtarget T4254:=[[55.000012,30.018711,40.750321],[1.000000,0.000000,0.000000,0.000000],[0,0,-1,0],[9E+09,9E+09,9E+09,9E+09,9E+09,9E+09]];
    CONST robtarget T4255:=[[55.000012,58.841502,40.750321],[1.000000,0.000000,0.000000,0.000000],[0,0,-1,0],[9E+09,9E+09,9E+09,9E+09,9E+09,9E+09]];
    CONST robtarget T4256:=[[53.500006,58.762255,40.750321],[1.000000,0.000000,0.000000,0.000000],[0,0,-1,0],[9E+09,9E+09,9E+09,9E+09,9E+09,9E+09]];
    CONST robtarget T4257:=[[53.500006,30.483202,40.750321],[1.000000,0.000000,0.000000,0.000000],[0,0,-1,0],[9E+09,9E+09,9E+09,9E+09,9E+09,9E+09]];
    CONST robtarget T4258:=[[52.000000,33.123088,40.750321],[1.000000,0.000000,0.000000,0.000000],[0,0,-1,0],[9E+09,9E+09,9E+09,9E+09,9E+09,9E+09]];
    CONST robtarget T4259:=[[52.000000,58.535318,40.750321],[1.000000,0.000000,0.000000,0.000000],[0,0,-1,0],[9E+09,9E+09,9E+09,9E+09,9E+09,9E+09]];
    CONST robtarget T4260:=[[50.499994,58.096460,40.750321],[1.000000,0.000000,0.000000,0.000000],[0,0,-1,0],[9E+09,9E+09,9E+09,9E+09,9E+09,9E+09]];
    CONST robtarget T4261:=[[50.499994,37.166186,40.750321],[1.000000,0.000000,0.000000,0.000000],[0,0,-1,0],[9E+09,9E+09,9E+09,9E+09,9E+09,9E+09]];
    CONST robtarget T4262:=[[48.999988,38.408162,40.750321],[1.000000,0.000000,0.000000,0.000000],[0,0,-1,0],[9E+09,9E+09,9E+09,9E+09,9E+09,9E+09]];
    CONST robtarget T4263:=[[48.999988,57.345139,40.750321],[1.000000,0.000000,0.000000,0.000000],[0,0,-1,0],[9E+09,9E+09,9E+09,9E+09,9E+09,9E+09]];
    CONST robtarget T4264:=[[47.499982,56.300306,40.750321],[1.000000,0.000000,0.000000,0.000000],[0,0,-1,0],[9E+09,9E+09,9E+09,9E+09,9E+09,9E+09]];
    CONST robtarget T4265:=[[47.499982,39.555172,40.750321],[1.000000,0.000000,0.000000,0.000000],[0,0,-1,0],[9E+09,9E+09,9E+09,9E+09,9E+09,9E+09]];
    CONST robtarget T4266:=[[45.999976,41.154240,40.750321],[1.000000,0.000000,0.000000,0.000000],[0,0,-1,0],[9E+09,9E+09,9E+09,9E+09,9E+09,9E+09]];
    CONST robtarget T4267:=[[45.999976,54.938672,40.750321],[1.000000,0.000000,0.000000,0.000000],[0,0,-1,0],[9E+09,9E+09,9E+09,9E+09,9E+09,9E+09]];
    CONST robtarget T4268:=[[44.499970,52.723926,40.750321],[1.000000,0.000000,0.000000,0.000000],[0,0,-1,0],[9E+09,9E+09,9E+09,9E+09,9E+09,9E+09]];
    CONST robtarget T4269:=[[44.499970,42.646312,40.750321],[1.000000,0.000000,0.000000,0.000000],[0,0,-1,0],[9E+09,9E+09,9E+09,9E+09,9E+09,9E+09]];
    CONST robtarget T4270:=[[42.999964,43.826022,40.750321],[1.000000,0.000000,0.000000,0.000000],[0,0,-1,0],[9E+09,9E+09,9E+09,9E+09,9E+09,9E+09]];
    CONST robtarget T4271:=[[42.999964,49.731638,40.750321],[1.000000,0.000000,0.000000,0.000000],[0,0,-1,0],[9E+09,9E+09,9E+09,9E+09,9E+09,9E+09]];
    CONST robtarget T4272:=[[42.999961,43.892572,41.250331],[1.000000,0.000000,0.000000,0.000000],[0,0,-1,0],[9E+09,9E+09,9E+09,9E+09,9E+09,9E+09]];
    CONST robtarget T4273:=[[42.999961,49.361580,41.250331],[1.000000,0.000000,0.000000,0.000000],[0,0,-1,0],[9E+09,9E+09,9E+09,9E+09,9E+09,9E+09]];
    CONST robtarget T4274:=[[42.999961,43.892572,41.250331],[1.000000,0.000000,0.000000,0.000000],[0,0,-1,0],[9E+09,9E+09,9E+09,9E+09,9E+09,9E+09]];
    CONST robtarget T4275:=[[42.999961,49.361580,41.250331],[1.000000,0.000000,0.000000,0.000000],[0,0,-1,0],[9E+09,9E+09,9E+09,9E+09,9E+09,9E+09]];
    CONST robtarget T4276:=[[44.499967,52.628460,41.250331],[1.000000,0.000000,0.000000,0.000000],[0,0,-1,0],[9E+09,9E+09,9E+09,9E+09,9E+09,9E+09]];
    CONST robtarget T4277:=[[44.499967,42.852661,41.250331],[1.000000,0.000000,0.000000,0.000000],[0,0,-1,0],[9E+09,9E+09,9E+09,9E+09,9E+09,9E+09]];
    CONST robtarget T4278:=[[45.999973,41.434647,41.250331],[1.000000,0.000000,0.000000,0.000000],[0,0,-1,0],[9E+09,9E+09,9E+09,9E+09,9E+09,9E+09]];
    CONST robtarget T4279:=[[45.999973,54.777961,41.250331],[1.000000,0.000000,0.000000,0.000000],[0,0,-1,0],[9E+09,9E+09,9E+09,9E+09,9E+09,9E+09]];
    CONST robtarget T4280:=[[47.499979,56.182009,41.250331],[1.000000,0.000000,0.000000,0.000000],[0,0,-1,0],[9E+09,9E+09,9E+09,9E+09,9E+09,9E+09]];
    CONST robtarget T4281:=[[47.499979,39.836843,41.250331],[1.000000,0.000000,0.000000,0.000000],[0,0,-1,0],[9E+09,9E+09,9E+09,9E+09,9E+09,9E+09]];
    CONST robtarget T4282:=[[48.999985,38.572340,41.250331],[1.000000,0.000000,0.000000,0.000000],[0,0,-1,0],[9E+09,9E+09,9E+09,9E+09,9E+09,9E+09]];
    CONST robtarget T4283:=[[48.999985,57.216424,41.250331],[1.000000,0.000000,0.000000,0.000000],[0,0,-1,0],[9E+09,9E+09,9E+09,9E+09,9E+09,9E+09]];
    CONST robtarget T4284:=[[50.499991,58.050029,41.250331],[1.000000,0.000000,0.000000,0.000000],[0,0,-1,0],[9E+09,9E+09,9E+09,9E+09,9E+09,9E+09]];
    CONST robtarget T4285:=[[50.499991,37.623125,41.250331],[1.000000,0.000000,0.000000,0.000000],[0,0,-1,0],[9E+09,9E+09,9E+09,9E+09,9E+09,9E+09]];
    CONST robtarget T4286:=[[51.999997,34.547257,41.250331],[1.000000,0.000000,0.000000,0.000000],[0,0,-1,0],[9E+09,9E+09,9E+09,9E+09,9E+09,9E+09]];
    CONST robtarget T4287:=[[51.999997,58.449384,41.250331],[1.000000,0.000000,0.000000,0.000000],[0,0,-1,0],[9E+09,9E+09,9E+09,9E+09,9E+09,9E+09]];
    CONST robtarget T4288:=[[53.500003,58.667944,41.250331],[1.000000,0.000000,0.000000,0.000000],[0,0,-1,0],[9E+09,9E+09,9E+09,9E+09,9E+09,9E+09]];
    CONST robtarget T4289:=[[53.500003,30.631761,41.250331],[1.000000,0.000000,0.000000,0.000000],[0,0,-1,0],[9E+09,9E+09,9E+09,9E+09,9E+09,9E+09]];
    CONST robtarget T4290:=[[55.000009,30.069203,41.250331],[1.000000,0.000000,0.000000,0.000000],[0,0,-1,0],[9E+09,9E+09,9E+09,9E+09,9E+09,9E+09]];
    CONST robtarget T4291:=[[55.000009,58.747191,41.250331],[1.000000,0.000000,0.000000,0.000000],[0,0,-1,0],[9E+09,9E+09,9E+09,9E+09,9E+09,9E+09]];
    CONST robtarget T4292:=[[56.500015,58.667944,41.250331],[1.000000,0.000000,0.000000,0.000000],[0,0,-1,0],[9E+09,9E+09,9E+09,9E+09,9E+09,9E+09]];
    CONST robtarget T4293:=[[56.500015,30.631764,41.250331],[1.000000,0.000000,0.000000,0.000000],[0,0,-1,0],[9E+09,9E+09,9E+09,9E+09,9E+09,9E+09]];
    CONST robtarget T4294:=[[58.000021,34.547269,41.250331],[1.000000,0.000000,0.000000,0.000000],[0,0,-1,0],[9E+09,9E+09,9E+09,9E+09,9E+09,9E+09]];
    CONST robtarget T4295:=[[58.000021,58.449383,41.250331],[1.000000,0.000000,0.000000,0.000000],[0,0,-1,0],[9E+09,9E+09,9E+09,9E+09,9E+09,9E+09]];
    CONST robtarget T4296:=[[59.500027,58.050028,41.250331],[1.000000,0.000000,0.000000,0.000000],[0,0,-1,0],[9E+09,9E+09,9E+09,9E+09,9E+09,9E+09]];
    CONST robtarget T4297:=[[59.500027,37.623128,41.250331],[1.000000,0.000000,0.000000,0.000000],[0,0,-1,0],[9E+09,9E+09,9E+09,9E+09,9E+09,9E+09]];
    CONST robtarget T4298:=[[61.000033,38.572343,41.250331],[1.000000,0.000000,0.000000,0.000000],[0,0,-1,0],[9E+09,9E+09,9E+09,9E+09,9E+09,9E+09]];
    CONST robtarget T4299:=[[61.000033,57.216422,41.250331],[1.000000,0.000000,0.000000,0.000000],[0,0,-1,0],[9E+09,9E+09,9E+09,9E+09,9E+09,9E+09]];
    CONST robtarget T4300:=[[62.500039,56.182005,41.250331],[1.000000,0.000000,0.000000,0.000000],[0,0,-1,0],[9E+09,9E+09,9E+09,9E+09,9E+09,9E+09]];
    CONST robtarget T4301:=[[62.500039,39.836847,41.250331],[1.000000,0.000000,0.000000,0.000000],[0,0,-1,0],[9E+09,9E+09,9E+09,9E+09,9E+09,9E+09]];
    CONST robtarget T4302:=[[64.000045,41.434651,41.250331],[1.000000,0.000000,0.000000,0.000000],[0,0,-1,0],[9E+09,9E+09,9E+09,9E+09,9E+09,9E+09]];
    CONST robtarget T4303:=[[64.000045,54.777958,41.250331],[1.000000,0.000000,0.000000,0.000000],[0,0,-1,0],[9E+09,9E+09,9E+09,9E+09,9E+09,9E+09]];
    CONST robtarget T4304:=[[65.500051,52.628454,41.250331],[1.000000,0.000000,0.000000,0.000000],[0,0,-1,0],[9E+09,9E+09,9E+09,9E+09,9E+09,9E+09]];
    CONST robtarget T4305:=[[65.500051,42.852675,41.250331],[1.000000,0.000000,0.000000,0.000000],[0,0,-1,0],[9E+09,9E+09,9E+09,9E+09,9E+09,9E+09]];
    CONST robtarget T4306:=[[67.000057,43.892581,41.250331],[1.000000,0.000000,0.000000,0.000000],[0,0,-1,0],[9E+09,9E+09,9E+09,9E+09,9E+09,9E+09]];
    CONST robtarget T4307:=[[67.000057,49.361569,41.250331],[1.000000,0.000000,0.000000,0.000000],[0,0,-1,0],[9E+09,9E+09,9E+09,9E+09,9E+09,9E+09]];
    CONST robtarget T4308:=[[67.000057,44.402616,41.750341],[1.000000,0.000000,0.000000,0.000000],[0,0,-1,0],[9E+09,9E+09,9E+09,9E+09,9E+09,9E+09]];
    CONST robtarget T4309:=[[67.000057,48.991522,41.750341],[1.000000,0.000000,0.000000,0.000000],[0,0,-1,0],[9E+09,9E+09,9E+09,9E+09,9E+09,9E+09]];
    CONST robtarget T4310:=[[67.000057,44.402616,41.750341],[1.000000,0.000000,0.000000,0.000000],[0,0,-1,0],[9E+09,9E+09,9E+09,9E+09,9E+09,9E+09]];
    CONST robtarget T4311:=[[67.000057,48.991522,41.750341],[1.000000,0.000000,0.000000,0.000000],[0,0,-1,0],[9E+09,9E+09,9E+09,9E+09,9E+09,9E+09]];
    CONST robtarget T4312:=[[65.500051,52.268733,41.750341],[1.000000,0.000000,0.000000,0.000000],[0,0,-1,0],[9E+09,9E+09,9E+09,9E+09,9E+09,9E+09]];
    CONST robtarget T4313:=[[65.500051,43.237915,41.750341],[1.000000,0.000000,0.000000,0.000000],[0,0,-1,0],[9E+09,9E+09,9E+09,9E+09,9E+09,9E+09]];
    CONST robtarget T4314:=[[64.000045,41.709401,41.750341],[1.000000,0.000000,0.000000,0.000000],[0,0,-1,0],[9E+09,9E+09,9E+09,9E+09,9E+09,9E+09]];
    CONST robtarget T4315:=[[64.000045,54.560067,41.750341],[1.000000,0.000000,0.000000,0.000000],[0,0,-1,0],[9E+09,9E+09,9E+09,9E+09,9E+09,9E+09]];
    CONST robtarget T4316:=[[62.500039,56.063713,41.750341],[1.000000,0.000000,0.000000,0.000000],[0,0,-1,0],[9E+09,9E+09,9E+09,9E+09,9E+09,9E+09]];
    CONST robtarget T4317:=[[62.500039,40.105231,41.750341],[1.000000,0.000000,0.000000,0.000000],[0,0,-1,0],[9E+09,9E+09,9E+09,9E+09,9E+09,9E+09]];
    CONST robtarget T4318:=[[61.000033,38.796618,41.750341],[1.000000,0.000000,0.000000,0.000000],[0,0,-1,0],[9E+09,9E+09,9E+09,9E+09,9E+09,9E+09]];
    CONST robtarget T4319:=[[61.000033,57.087709,41.750341],[1.000000,0.000000,0.000000,0.000000],[0,0,-1,0],[9E+09,9E+09,9E+09,9E+09,9E+09,9E+09]];
    CONST robtarget T4320:=[[59.500027,57.973629,41.750341],[1.000000,0.000000,0.000000,0.000000],[0,0,-1,0],[9E+09,9E+09,9E+09,9E+09,9E+09,9E+09]];
    CONST robtarget T4321:=[[59.500027,37.822308,41.750341],[1.000000,0.000000,0.000000,0.000000],[0,0,-1,0],[9E+09,9E+09,9E+09,9E+09,9E+09,9E+09]];
    CONST robtarget T4322:=[[58.000021,35.796954,41.750341],[1.000000,0.000000,0.000000,0.000000],[0,0,-1,0],[9E+09,9E+09,9E+09,9E+09,9E+09,9E+09]];
    CONST robtarget T4323:=[[58.000021,58.309653,41.750341],[1.000000,0.000000,0.000000,0.000000],[0,0,-1,0],[9E+09,9E+09,9E+09,9E+09,9E+09,9E+09]];
    CONST robtarget T4324:=[[56.500015,58.575026,41.750341],[1.000000,0.000000,0.000000,0.000000],[0,0,-1,0],[9E+09,9E+09,9E+09,9E+09,9E+09,9E+09]];
    CONST robtarget T4325:=[[56.500015,33.270380,41.750341],[1.000000,0.000000,0.000000,0.000000],[0,0,-1,0],[9E+09,9E+09,9E+09,9E+09,9E+09,9E+09]];
    CONST robtarget T4326:=[[55.000009,30.362363,41.750341],[1.000000,0.000000,0.000000,0.000000],[0,0,-1,0],[9E+09,9E+09,9E+09,9E+09,9E+09,9E+09]];
    CONST robtarget T4327:=[[55.000009,58.652880,41.750341],[1.000000,0.000000,0.000000,0.000000],[0,0,-1,0],[9E+09,9E+09,9E+09,9E+09,9E+09,9E+09]];
    CONST robtarget T4328:=[[53.500003,58.575026,41.750341],[1.000000,0.000000,0.000000,0.000000],[0,0,-1,0],[9E+09,9E+09,9E+09,9E+09,9E+09,9E+09]];
    CONST robtarget T4329:=[[53.500003,33.270377,41.750341],[1.000000,0.000000,0.000000,0.000000],[0,0,-1,0],[9E+09,9E+09,9E+09,9E+09,9E+09,9E+09]];
    CONST robtarget T4330:=[[51.999997,35.796947,41.750341],[1.000000,0.000000,0.000000,0.000000],[0,0,-1,0],[9E+09,9E+09,9E+09,9E+09,9E+09,9E+09]];
    CONST robtarget T4331:=[[51.999997,58.309654,41.750341],[1.000000,0.000000,0.000000,0.000000],[0,0,-1,0],[9E+09,9E+09,9E+09,9E+09,9E+09,9E+09]];
    CONST robtarget T4332:=[[50.499991,57.973630,41.750341],[1.000000,0.000000,0.000000,0.000000],[0,0,-1,0],[9E+09,9E+09,9E+09,9E+09,9E+09,9E+09]];
    CONST robtarget T4333:=[[50.499991,37.822306,41.750341],[1.000000,0.000000,0.000000,0.000000],[0,0,-1,0],[9E+09,9E+09,9E+09,9E+09,9E+09,9E+09]];
    CONST robtarget T4334:=[[48.999985,38.796617,41.750341],[1.000000,0.000000,0.000000,0.000000],[0,0,-1,0],[9E+09,9E+09,9E+09,9E+09,9E+09,9E+09]];
    CONST robtarget T4335:=[[48.999985,57.087711,41.750341],[1.000000,0.000000,0.000000,0.000000],[0,0,-1,0],[9E+09,9E+09,9E+09,9E+09,9E+09,9E+09]];
    CONST robtarget T4336:=[[47.499979,56.063716,41.750341],[1.000000,0.000000,0.000000,0.000000],[0,0,-1,0],[9E+09,9E+09,9E+09,9E+09,9E+09,9E+09]];
    CONST robtarget T4337:=[[47.499979,40.105228,41.750341],[1.000000,0.000000,0.000000,0.000000],[0,0,-1,0],[9E+09,9E+09,9E+09,9E+09,9E+09,9E+09]];
    CONST robtarget T4338:=[[45.999973,41.709399,41.750341],[1.000000,0.000000,0.000000,0.000000],[0,0,-1,0],[9E+09,9E+09,9E+09,9E+09,9E+09,9E+09]];
    CONST robtarget T4339:=[[45.999973,54.560070,41.750341],[1.000000,0.000000,0.000000,0.000000],[0,0,-1,0],[9E+09,9E+09,9E+09,9E+09,9E+09,9E+09]];
    CONST robtarget T4340:=[[44.499967,52.268737,41.750341],[1.000000,0.000000,0.000000,0.000000],[0,0,-1,0],[9E+09,9E+09,9E+09,9E+09,9E+09,9E+09]];
    CONST robtarget T4341:=[[44.499967,43.237914,41.750341],[1.000000,0.000000,0.000000,0.000000],[0,0,-1,0],[9E+09,9E+09,9E+09,9E+09,9E+09,9E+09]];
    CONST robtarget T4342:=[[42.999961,44.402616,41.750341],[1.000000,0.000000,0.000000,0.000000],[0,0,-1,0],[9E+09,9E+09,9E+09,9E+09,9E+09,9E+09]];
    CONST robtarget T4343:=[[42.999961,48.991530,41.750341],[1.000000,0.000000,0.000000,0.000000],[0,0,-1,0],[9E+09,9E+09,9E+09,9E+09,9E+09,9E+09]];
    CONST robtarget T4344:=[[42.999959,44.998836,42.250351],[1.000000,0.000000,0.000000,0.000000],[0,0,-1,0],[9E+09,9E+09,9E+09,9E+09,9E+09,9E+09]];
    CONST robtarget T4345:=[[42.999959,48.236902,42.250351],[1.000000,0.000000,0.000000,0.000000],[0,0,-1,0],[9E+09,9E+09,9E+09,9E+09,9E+09,9E+09]];
    CONST robtarget T4346:=[[42.999959,44.998836,42.250351],[1.000000,0.000000,0.000000,0.000000],[0,0,-1,0],[9E+09,9E+09,9E+09,9E+09,9E+09,9E+09]];
    CONST robtarget T4347:=[[42.999959,48.236902,42.250351],[1.000000,0.000000,0.000000,0.000000],[0,0,-1,0],[9E+09,9E+09,9E+09,9E+09,9E+09,9E+09]];
    CONST robtarget T4348:=[[44.499965,51.685384,42.250351],[1.000000,0.000000,0.000000,0.000000],[0,0,-1,0],[9E+09,9E+09,9E+09,9E+09,9E+09,9E+09]];
    CONST robtarget T4349:=[[44.499965,43.413939,42.250351],[1.000000,0.000000,0.000000,0.000000],[0,0,-1,0],[9E+09,9E+09,9E+09,9E+09,9E+09,9E+09]];
    CONST robtarget T4350:=[[45.999971,42.004912,42.250351],[1.000000,0.000000,0.000000,0.000000],[0,0,-1,0],[9E+09,9E+09,9E+09,9E+09,9E+09,9E+09]];
    CONST robtarget T4351:=[[45.999971,54.258910,42.250351],[1.000000,0.000000,0.000000,0.000000],[0,0,-1,0],[9E+09,9E+09,9E+09,9E+09,9E+09,9E+09]];
    CONST robtarget T4352:=[[47.499977,55.843542,42.250351],[1.000000,0.000000,0.000000,0.000000],[0,0,-1,0],[9E+09,9E+09,9E+09,9E+09,9E+09,9E+09]];
    CONST robtarget T4353:=[[47.499977,40.371383,42.250351],[1.000000,0.000000,0.000000,0.000000],[0,0,-1,0],[9E+09,9E+09,9E+09,9E+09,9E+09,9E+09]];
    CONST robtarget T4354:=[[48.999983,39.023252,42.250351],[1.000000,0.000000,0.000000,0.000000],[0,0,-1,0],[9E+09,9E+09,9E+09,9E+09,9E+09,9E+09]];
    CONST robtarget T4355:=[[48.999983,56.958997,42.250351],[1.000000,0.000000,0.000000,0.000000],[0,0,-1,0],[9E+09,9E+09,9E+09,9E+09,9E+09,9E+09]];
    CONST robtarget T4356:=[[50.499989,57.760230,42.250351],[1.000000,0.000000,0.000000,0.000000],[0,0,-1,0],[9E+09,9E+09,9E+09,9E+09,9E+09,9E+09]];
    CONST robtarget T4357:=[[50.499989,38.015537,42.250351],[1.000000,0.000000,0.000000,0.000000],[0,0,-1,0],[9E+09,9E+09,9E+09,9E+09,9E+09,9E+09]];
    CONST robtarget T4358:=[[51.999995,36.847447,42.250351],[1.000000,0.000000,0.000000,0.000000],[0,0,-1,0],[9E+09,9E+09,9E+09,9E+09,9E+09,9E+09]];
    CONST robtarget T4359:=[[51.999995,58.171618,42.250351],[1.000000,0.000000,0.000000,0.000000],[0,0,-1,0],[9E+09,9E+09,9E+09,9E+09,9E+09,9E+09]];
    CONST robtarget T4360:=[[53.500001,58.477413,42.250351],[1.000000,0.000000,0.000000,0.000000],[0,0,-1,0],[9E+09,9E+09,9E+09,9E+09,9E+09,9E+09]];
    CONST robtarget T4361:=[[53.500001,34.996948,42.250351],[1.000000,0.000000,0.000000,0.000000],[0,0,-1,0],[9E+09,9E+09,9E+09,9E+09,9E+09,9E+09]];
    CONST robtarget T4362:=[[55.000007,34.716682,42.250351],[1.000000,0.000000,0.000000,0.000000],[0,0,-1,0],[9E+09,9E+09,9E+09,9E+09,9E+09,9E+09]];
    CONST robtarget T4363:=[[55.000007,58.553746,42.250351],[1.000000,0.000000,0.000000,0.000000],[0,0,-1,0],[9E+09,9E+09,9E+09,9E+09,9E+09,9E+09]];
    CONST robtarget T4364:=[[56.500013,58.477412,42.250351],[1.000000,0.000000,0.000000,0.000000],[0,0,-1,0],[9E+09,9E+09,9E+09,9E+09,9E+09,9E+09]];
    CONST robtarget T4365:=[[56.500013,34.996948,42.250351],[1.000000,0.000000,0.000000,0.000000],[0,0,-1,0],[9E+09,9E+09,9E+09,9E+09,9E+09,9E+09]];
    CONST robtarget T4366:=[[58.000019,36.847448,42.250351],[1.000000,0.000000,0.000000,0.000000],[0,0,-1,0],[9E+09,9E+09,9E+09,9E+09,9E+09,9E+09]];
    CONST robtarget T4367:=[[58.000019,58.171618,42.250351],[1.000000,0.000000,0.000000,0.000000],[0,0,-1,0],[9E+09,9E+09,9E+09,9E+09,9E+09,9E+09]];
    CONST robtarget T4368:=[[59.500025,57.760230,42.250351],[1.000000,0.000000,0.000000,0.000000],[0,0,-1,0],[9E+09,9E+09,9E+09,9E+09,9E+09,9E+09]];
    CONST robtarget T4369:=[[59.500025,38.015537,42.250351],[1.000000,0.000000,0.000000,0.000000],[0,0,-1,0],[9E+09,9E+09,9E+09,9E+09,9E+09,9E+09]];
    CONST robtarget T4370:=[[61.000031,39.023252,42.250351],[1.000000,0.000000,0.000000,0.000000],[0,0,-1,0],[9E+09,9E+09,9E+09,9E+09,9E+09,9E+09]];
    CONST robtarget T4371:=[[61.000031,56.958996,42.250351],[1.000000,0.000000,0.000000,0.000000],[0,0,-1,0],[9E+09,9E+09,9E+09,9E+09,9E+09,9E+09]];
    CONST robtarget T4372:=[[62.500037,55.843542,42.250351],[1.000000,0.000000,0.000000,0.000000],[0,0,-1,0],[9E+09,9E+09,9E+09,9E+09,9E+09,9E+09]];
    CONST robtarget T4373:=[[62.500037,40.371384,42.250351],[1.000000,0.000000,0.000000,0.000000],[0,0,-1,0],[9E+09,9E+09,9E+09,9E+09,9E+09,9E+09]];
    CONST robtarget T4374:=[[64.000043,42.004912,42.250351],[1.000000,0.000000,0.000000,0.000000],[0,0,-1,0],[9E+09,9E+09,9E+09,9E+09,9E+09,9E+09]];
    CONST robtarget T4375:=[[64.000043,54.258911,42.250351],[1.000000,0.000000,0.000000,0.000000],[0,0,-1,0],[9E+09,9E+09,9E+09,9E+09,9E+09,9E+09]];
    CONST robtarget T4376:=[[65.500049,51.685384,42.250351],[1.000000,0.000000,0.000000,0.000000],[0,0,-1,0],[9E+09,9E+09,9E+09,9E+09,9E+09,9E+09]];
    CONST robtarget T4377:=[[65.500049,43.413939,42.250351],[1.000000,0.000000,0.000000,0.000000],[0,0,-1,0],[9E+09,9E+09,9E+09,9E+09,9E+09,9E+09]];
    CONST robtarget T4378:=[[67.000055,44.998837,42.250351],[1.000000,0.000000,0.000000,0.000000],[0,0,-1,0],[9E+09,9E+09,9E+09,9E+09,9E+09,9E+09]];
    CONST robtarget T4379:=[[67.000055,48.236902,42.250351],[1.000000,0.000000,0.000000,0.000000],[0,0,-1,0],[9E+09,9E+09,9E+09,9E+09,9E+09,9E+09]];
    CONST robtarget T4380:=[[66.250052,44.221433,42.750361],[1.000000,0.000000,0.000000,0.000000],[0,0,-1,0],[9E+09,9E+09,9E+09,9E+09,9E+09,9E+09]];
    CONST robtarget T4381:=[[66.250052,49.472574,42.750361],[1.000000,0.000000,0.000000,0.000000],[0,0,-1,0],[9E+09,9E+09,9E+09,9E+09,9E+09,9E+09]];
    CONST robtarget T4382:=[[66.250052,44.221433,42.750361],[1.000000,0.000000,0.000000,0.000000],[0,0,-1,0],[9E+09,9E+09,9E+09,9E+09,9E+09,9E+09]];
    CONST robtarget T4383:=[[66.250052,49.472574,42.750361],[1.000000,0.000000,0.000000,0.000000],[0,0,-1,0],[9E+09,9E+09,9E+09,9E+09,9E+09,9E+09]];
    CONST robtarget T4384:=[[64.750046,52.608003,42.750361],[1.000000,0.000000,0.000000,0.000000],[0,0,-1,0],[9E+09,9E+09,9E+09,9E+09,9E+09,9E+09]];
    CONST robtarget T4385:=[[64.750046,43.306281,42.750361],[1.000000,0.000000,0.000000,0.000000],[0,0,-1,0],[9E+09,9E+09,9E+09,9E+09,9E+09,9E+09]];
    CONST robtarget T4386:=[[63.250040,41.505974,42.750361],[1.000000,0.000000,0.000000,0.000000],[0,0,-1,0],[9E+09,9E+09,9E+09,9E+09,9E+09,9E+09]];
    CONST robtarget T4387:=[[63.250040,54.928906,42.750361],[1.000000,0.000000,0.000000,0.000000],[0,0,-1,0],[9E+09,9E+09,9E+09,9E+09,9E+09,9E+09]];
    CONST robtarget T4388:=[[61.750034,56.271779,42.750361],[1.000000,0.000000,0.000000,0.000000],[0,0,-1,0],[9E+09,9E+09,9E+09,9E+09,9E+09,9E+09]];
    CONST robtarget T4389:=[[61.750034,39.993766,42.750361],[1.000000,0.000000,0.000000,0.000000],[0,0,-1,0],[9E+09,9E+09,9E+09,9E+09,9E+09,9E+09]];
    CONST robtarget T4390:=[[60.250028,38.725118,42.750361],[1.000000,0.000000,0.000000,0.000000],[0,0,-1,0],[9E+09,9E+09,9E+09,9E+09,9E+09,9E+09]];
    CONST robtarget T4391:=[[60.250028,57.224212,42.750361],[1.000000,0.000000,0.000000,0.000000],[0,0,-1,0],[9E+09,9E+09,9E+09,9E+09,9E+09,9E+09]];
    CONST robtarget T4392:=[[58.750022,57.869448,42.750361],[1.000000,0.000000,0.000000,0.000000],[0,0,-1,0],[9E+09,9E+09,9E+09,9E+09,9E+09,9E+09]];
    CONST robtarget T4393:=[[58.750022,37.851516,42.750361],[1.000000,0.000000,0.000000,0.000000],[0,0,-1,0],[9E+09,9E+09,9E+09,9E+09,9E+09,9E+09]];
    CONST robtarget T4394:=[[57.250016,36.656739,42.750361],[1.000000,0.000000,0.000000,0.000000],[0,0,-1,0],[9E+09,9E+09,9E+09,9E+09,9E+09,9E+09]];
    CONST robtarget T4395:=[[57.250016,58.191331,42.750361],[1.000000,0.000000,0.000000,0.000000],[0,0,-1,0],[9E+09,9E+09,9E+09,9E+09,9E+09,9E+09]];
    CONST robtarget T4396:=[[55.750010,58.325833,42.750361],[1.000000,0.000000,0.000000,0.000000],[0,0,-1,0],[9E+09,9E+09,9E+09,9E+09,9E+09,9E+09]];
    CONST robtarget T4397:=[[55.750010,35.788946,42.750361],[1.000000,0.000000,0.000000,0.000000],[0,0,-1,0],[9E+09,9E+09,9E+09,9E+09,9E+09,9E+09]];
    CONST robtarget T4398:=[[54.250004,35.788946,42.750361],[1.000000,0.000000,0.000000,0.000000],[0,0,-1,0],[9E+09,9E+09,9E+09,9E+09,9E+09,9E+09]];
    CONST robtarget T4399:=[[54.250004,58.325833,42.750361],[1.000000,0.000000,0.000000,0.000000],[0,0,-1,0],[9E+09,9E+09,9E+09,9E+09,9E+09,9E+09]];
    CONST robtarget T4400:=[[52.749998,58.191331,42.750361],[1.000000,0.000000,0.000000,0.000000],[0,0,-1,0],[9E+09,9E+09,9E+09,9E+09,9E+09,9E+09]];
    CONST robtarget T4401:=[[52.749998,36.656739,42.750361],[1.000000,0.000000,0.000000,0.000000],[0,0,-1,0],[9E+09,9E+09,9E+09,9E+09,9E+09,9E+09]];
    CONST robtarget T4402:=[[51.249992,37.851516,42.750361],[1.000000,0.000000,0.000000,0.000000],[0,0,-1,0],[9E+09,9E+09,9E+09,9E+09,9E+09,9E+09]];
    CONST robtarget T4403:=[[51.249992,57.869448,42.750361],[1.000000,0.000000,0.000000,0.000000],[0,0,-1,0],[9E+09,9E+09,9E+09,9E+09,9E+09,9E+09]];
    CONST robtarget T4404:=[[49.749986,57.224212,42.750361],[1.000000,0.000000,0.000000,0.000000],[0,0,-1,0],[9E+09,9E+09,9E+09,9E+09,9E+09,9E+09]];
    CONST robtarget T4405:=[[49.749986,38.725118,42.750361],[1.000000,0.000000,0.000000,0.000000],[0,0,-1,0],[9E+09,9E+09,9E+09,9E+09,9E+09,9E+09]];
    CONST robtarget T4406:=[[48.249980,39.993770,42.750361],[1.000000,0.000000,0.000000,0.000000],[0,0,-1,0],[9E+09,9E+09,9E+09,9E+09,9E+09,9E+09]];
    CONST robtarget T4407:=[[48.249980,56.271780,42.750361],[1.000000,0.000000,0.000000,0.000000],[0,0,-1,0],[9E+09,9E+09,9E+09,9E+09,9E+09,9E+09]];
    CONST robtarget T4408:=[[46.749974,54.928905,42.750361],[1.000000,0.000000,0.000000,0.000000],[0,0,-1,0],[9E+09,9E+09,9E+09,9E+09,9E+09,9E+09]];
    CONST robtarget T4409:=[[46.749974,41.505975,42.750361],[1.000000,0.000000,0.000000,0.000000],[0,0,-1,0],[9E+09,9E+09,9E+09,9E+09,9E+09,9E+09]];
    CONST robtarget T4410:=[[45.249968,43.306281,42.750361],[1.000000,0.000000,0.000000,0.000000],[0,0,-1,0],[9E+09,9E+09,9E+09,9E+09,9E+09,9E+09]];
    CONST robtarget T4411:=[[45.249968,52.608002,42.750361],[1.000000,0.000000,0.000000,0.000000],[0,0,-1,0],[9E+09,9E+09,9E+09,9E+09,9E+09,9E+09]];
    CONST robtarget T4412:=[[43.749962,49.472574,42.750361],[1.000000,0.000000,0.000000,0.000000],[0,0,-1,0],[9E+09,9E+09,9E+09,9E+09,9E+09,9E+09]];
    CONST robtarget T4413:=[[43.749962,44.221443,42.750361],[1.000000,0.000000,0.000000,0.000000],[0,0,-1,0],[9E+09,9E+09,9E+09,9E+09,9E+09,9E+09]];
    CONST robtarget T4414:=[[44.499965,44.249106,43.250371],[1.000000,0.000000,0.000000,0.000000],[0,0,-1,0],[9E+09,9E+09,9E+09,9E+09,9E+09,9E+09]];
    CONST robtarget T4415:=[[44.499965,50.424926,43.250371],[1.000000,0.000000,0.000000,0.000000],[0,0,-1,0],[9E+09,9E+09,9E+09,9E+09,9E+09,9E+09]];
    CONST robtarget T4416:=[[44.499965,44.249106,43.250371],[1.000000,0.000000,0.000000,0.000000],[0,0,-1,0],[9E+09,9E+09,9E+09,9E+09,9E+09,9E+09]];
    CONST robtarget T4417:=[[44.499965,50.424926,43.250371],[1.000000,0.000000,0.000000,0.000000],[0,0,-1,0],[9E+09,9E+09,9E+09,9E+09,9E+09,9E+09]];
    CONST robtarget T4418:=[[45.999971,53.377281,43.250371],[1.000000,0.000000,0.000000,0.000000],[0,0,-1,0],[9E+09,9E+09,9E+09,9E+09,9E+09,9E+09]];
    CONST robtarget T4419:=[[45.999971,42.773348,43.250371],[1.000000,0.000000,0.000000,0.000000],[0,0,-1,0],[9E+09,9E+09,9E+09,9E+09,9E+09,9E+09]];
    CONST robtarget T4420:=[[47.499977,41.115132,43.250371],[1.000000,0.000000,0.000000,0.000000],[0,0,-1,0],[9E+09,9E+09,9E+09,9E+09,9E+09,9E+09]];
    CONST robtarget T4421:=[[47.499977,55.302933,43.250371],[1.000000,0.000000,0.000000,0.000000],[0,0,-1,0],[9E+09,9E+09,9E+09,9E+09,9E+09,9E+09]];
    CONST robtarget T4422:=[[48.999983,56.679781,43.250371],[1.000000,0.000000,0.000000,0.000000],[0,0,-1,0],[9E+09,9E+09,9E+09,9E+09,9E+09,9E+09]];
    CONST robtarget T4423:=[[48.999983,39.641897,43.250371],[1.000000,0.000000,0.000000,0.000000],[0,0,-1,0],[9E+09,9E+09,9E+09,9E+09,9E+09,9E+09]];
    CONST robtarget T4424:=[[50.499989,38.573807,43.250371],[1.000000,0.000000,0.000000,0.000000],[0,0,-1,0],[9E+09,9E+09,9E+09,9E+09,9E+09,9E+09]];
    CONST robtarget T4425:=[[50.499989,57.333692,43.250371],[1.000000,0.000000,0.000000,0.000000],[0,0,-1,0],[9E+09,9E+09,9E+09,9E+09,9E+09,9E+09]];
    CONST robtarget T4426:=[[51.999995,57.863303,43.250371],[1.000000,0.000000,0.000000,0.000000],[0,0,-1,0],[9E+09,9E+09,9E+09,9E+09,9E+09,9E+09]];
    CONST robtarget T4427:=[[51.999995,37.767749,43.250371],[1.000000,0.000000,0.000000,0.000000],[0,0,-1,0],[9E+09,9E+09,9E+09,9E+09,9E+09,9E+09]];
    CONST robtarget T4428:=[[53.500001,37.037102,43.250371],[1.000000,0.000000,0.000000,0.000000],[0,0,-1,0],[9E+09,9E+09,9E+09,9E+09,9E+09,9E+09]];
    CONST robtarget T4429:=[[53.500001,58.098140,43.250371],[1.000000,0.000000,0.000000,0.000000],[0,0,-1,0],[9E+09,9E+09,9E+09,9E+09,9E+09,9E+09]];
    CONST robtarget T4430:=[[55.000007,58.182798,43.250371],[1.000000,0.000000,0.000000,0.000000],[0,0,-1,0],[9E+09,9E+09,9E+09,9E+09,9E+09,9E+09]];
    CONST robtarget T4431:=[[55.000007,36.717480,43.250371],[1.000000,0.000000,0.000000,0.000000],[0,0,-1,0],[9E+09,9E+09,9E+09,9E+09,9E+09,9E+09]];
    CONST robtarget T4432:=[[56.500013,37.037101,43.250371],[1.000000,0.000000,0.000000,0.000000],[0,0,-1,0],[9E+09,9E+09,9E+09,9E+09,9E+09,9E+09]];
    CONST robtarget T4433:=[[56.500013,58.098140,43.250371],[1.000000,0.000000,0.000000,0.000000],[0,0,-1,0],[9E+09,9E+09,9E+09,9E+09,9E+09,9E+09]];
    CONST robtarget T4434:=[[58.000019,57.863303,43.250371],[1.000000,0.000000,0.000000,0.000000],[0,0,-1,0],[9E+09,9E+09,9E+09,9E+09,9E+09,9E+09]];
    CONST robtarget T4435:=[[58.000019,37.767748,43.250371],[1.000000,0.000000,0.000000,0.000000],[0,0,-1,0],[9E+09,9E+09,9E+09,9E+09,9E+09,9E+09]];
    CONST robtarget T4436:=[[59.500025,38.573811,43.250371],[1.000000,0.000000,0.000000,0.000000],[0,0,-1,0],[9E+09,9E+09,9E+09,9E+09,9E+09,9E+09]];
    CONST robtarget T4437:=[[59.500025,57.333692,43.250371],[1.000000,0.000000,0.000000,0.000000],[0,0,-1,0],[9E+09,9E+09,9E+09,9E+09,9E+09,9E+09]];
    CONST robtarget T4438:=[[61.000031,56.679780,43.250371],[1.000000,0.000000,0.000000,0.000000],[0,0,-1,0],[9E+09,9E+09,9E+09,9E+09,9E+09,9E+09]];
    CONST robtarget T4439:=[[61.000031,39.641891,43.250371],[1.000000,0.000000,0.000000,0.000000],[0,0,-1,0],[9E+09,9E+09,9E+09,9E+09,9E+09,9E+09]];
    CONST robtarget T4440:=[[62.500037,41.115128,43.250371],[1.000000,0.000000,0.000000,0.000000],[0,0,-1,0],[9E+09,9E+09,9E+09,9E+09,9E+09,9E+09]];
    CONST robtarget T4441:=[[62.500037,55.302934,43.250371],[1.000000,0.000000,0.000000,0.000000],[0,0,-1,0],[9E+09,9E+09,9E+09,9E+09,9E+09,9E+09]];
    CONST robtarget T4442:=[[64.000043,53.377283,43.250371],[1.000000,0.000000,0.000000,0.000000],[0,0,-1,0],[9E+09,9E+09,9E+09,9E+09,9E+09,9E+09]];
    CONST robtarget T4443:=[[64.000043,42.773348,43.250371],[1.000000,0.000000,0.000000,0.000000],[0,0,-1,0],[9E+09,9E+09,9E+09,9E+09,9E+09,9E+09]];
    CONST robtarget T4444:=[[65.500049,44.249106,43.250371],[1.000000,0.000000,0.000000,0.000000],[0,0,-1,0],[9E+09,9E+09,9E+09,9E+09,9E+09,9E+09]];
    CONST robtarget T4445:=[[65.500049,50.424928,43.250371],[1.000000,0.000000,0.000000,0.000000],[0,0,-1,0],[9E+09,9E+09,9E+09,9E+09,9E+09,9E+09]];
    CONST robtarget T4446:=[[65.500049,45.119837,43.750381],[1.000000,0.000000,0.000000,0.000000],[0,0,-1,0],[9E+09,9E+09,9E+09,9E+09,9E+09,9E+09]];
    CONST robtarget T4447:=[[65.500049,49.812885,43.750381],[1.000000,0.000000,0.000000,0.000000],[0,0,-1,0],[9E+09,9E+09,9E+09,9E+09,9E+09,9E+09]];
    CONST robtarget T4448:=[[65.500049,45.119837,43.750381],[1.000000,0.000000,0.000000,0.000000],[0,0,-1,0],[9E+09,9E+09,9E+09,9E+09,9E+09,9E+09]];
    CONST robtarget T4449:=[[65.500049,49.812885,43.750381],[1.000000,0.000000,0.000000,0.000000],[0,0,-1,0],[9E+09,9E+09,9E+09,9E+09,9E+09,9E+09]];
    CONST robtarget T4450:=[[64.000043,52.751074,43.750381],[1.000000,0.000000,0.000000,0.000000],[0,0,-1,0],[9E+09,9E+09,9E+09,9E+09,9E+09,9E+09]];
    CONST robtarget T4451:=[[64.000043,43.294101,43.750381],[1.000000,0.000000,0.000000,0.000000],[0,0,-1,0],[9E+09,9E+09,9E+09,9E+09,9E+09,9E+09]];
    CONST robtarget T4452:=[[62.500037,41.513575,43.750381],[1.000000,0.000000,0.000000,0.000000],[0,0,-1,0],[9E+09,9E+09,9E+09,9E+09,9E+09,9E+09]];
    CONST robtarget T4453:=[[62.500037,54.974258,43.750381],[1.000000,0.000000,0.000000,0.000000],[0,0,-1,0],[9E+09,9E+09,9E+09,9E+09,9E+09,9E+09]];
    CONST robtarget T4454:=[[61.000031,56.284612,43.750381],[1.000000,0.000000,0.000000,0.000000],[0,0,-1,0],[9E+09,9E+09,9E+09,9E+09,9E+09,9E+09]];
    CONST robtarget T4455:=[[61.000031,39.980402,43.750381],[1.000000,0.000000,0.000000,0.000000],[0,0,-1,0],[9E+09,9E+09,9E+09,9E+09,9E+09,9E+09]];
    CONST robtarget T4456:=[[59.500025,38.864453,43.750381],[1.000000,0.000000,0.000000,0.000000],[0,0,-1,0],[9E+09,9E+09,9E+09,9E+09,9E+09,9E+09]];
    CONST robtarget T4457:=[[59.500025,57.122334,43.750381],[1.000000,0.000000,0.000000,0.000000],[0,0,-1,0],[9E+09,9E+09,9E+09,9E+09,9E+09,9E+09]];
    CONST robtarget T4458:=[[58.000019,57.651620,43.750381],[1.000000,0.000000,0.000000,0.000000],[0,0,-1,0],[9E+09,9E+09,9E+09,9E+09,9E+09,9E+09]];
    CONST robtarget T4459:=[[58.000019,38.060967,43.750381],[1.000000,0.000000,0.000000,0.000000],[0,0,-1,0],[9E+09,9E+09,9E+09,9E+09,9E+09,9E+09]];
    CONST robtarget T4460:=[[56.500013,37.582886,43.750381],[1.000000,0.000000,0.000000,0.000000],[0,0,-1,0],[9E+09,9E+09,9E+09,9E+09,9E+09,9E+09]];
    CONST robtarget T4461:=[[56.500013,57.908504,43.750381],[1.000000,0.000000,0.000000,0.000000],[0,0,-1,0],[9E+09,9E+09,9E+09,9E+09,9E+09,9E+09]];
    CONST robtarget T4462:=[[55.000007,57.997324,43.750381],[1.000000,0.000000,0.000000,0.000000],[0,0,-1,0],[9E+09,9E+09,9E+09,9E+09,9E+09,9E+09]];
    CONST robtarget T4463:=[[55.000007,37.484561,43.750381],[1.000000,0.000000,0.000000,0.000000],[0,0,-1,0],[9E+09,9E+09,9E+09,9E+09,9E+09,9E+09]];
    CONST robtarget T4464:=[[53.500001,37.582886,43.750381],[1.000000,0.000000,0.000000,0.000000],[0,0,-1,0],[9E+09,9E+09,9E+09,9E+09,9E+09,9E+09]];
    CONST robtarget T4465:=[[53.500001,57.908504,43.750381],[1.000000,0.000000,0.000000,0.000000],[0,0,-1,0],[9E+09,9E+09,9E+09,9E+09,9E+09,9E+09]];
    CONST robtarget T4466:=[[51.999995,57.651620,43.750381],[1.000000,0.000000,0.000000,0.000000],[0,0,-1,0],[9E+09,9E+09,9E+09,9E+09,9E+09,9E+09]];
    CONST robtarget T4467:=[[51.999995,38.060967,43.750381],[1.000000,0.000000,0.000000,0.000000],[0,0,-1,0],[9E+09,9E+09,9E+09,9E+09,9E+09,9E+09]];
    CONST robtarget T4468:=[[50.499989,38.864447,43.750381],[1.000000,0.000000,0.000000,0.000000],[0,0,-1,0],[9E+09,9E+09,9E+09,9E+09,9E+09,9E+09]];
    CONST robtarget T4469:=[[50.499989,57.122334,43.750381],[1.000000,0.000000,0.000000,0.000000],[0,0,-1,0],[9E+09,9E+09,9E+09,9E+09,9E+09,9E+09]];
    CONST robtarget T4470:=[[48.999983,56.284613,43.750381],[1.000000,0.000000,0.000000,0.000000],[0,0,-1,0],[9E+09,9E+09,9E+09,9E+09,9E+09,9E+09]];
    CONST robtarget T4471:=[[48.999983,39.980411,43.750381],[1.000000,0.000000,0.000000,0.000000],[0,0,-1,0],[9E+09,9E+09,9E+09,9E+09,9E+09,9E+09]];
    CONST robtarget T4472:=[[47.499977,41.513576,43.750381],[1.000000,0.000000,0.000000,0.000000],[0,0,-1,0],[9E+09,9E+09,9E+09,9E+09,9E+09,9E+09]];
    CONST robtarget T4473:=[[47.499977,54.974259,43.750381],[1.000000,0.000000,0.000000,0.000000],[0,0,-1,0],[9E+09,9E+09,9E+09,9E+09,9E+09,9E+09]];
    CONST robtarget T4474:=[[45.999971,52.751074,43.750381],[1.000000,0.000000,0.000000,0.000000],[0,0,-1,0],[9E+09,9E+09,9E+09,9E+09,9E+09,9E+09]];
    CONST robtarget T4475:=[[45.999971,43.294100,43.750381],[1.000000,0.000000,0.000000,0.000000],[0,0,-1,0],[9E+09,9E+09,9E+09,9E+09,9E+09,9E+09]];
    CONST robtarget T4476:=[[44.499965,45.119837,43.750381],[1.000000,0.000000,0.000000,0.000000],[0,0,-1,0],[9E+09,9E+09,9E+09,9E+09,9E+09,9E+09]];
    CONST robtarget T4477:=[[44.499965,49.812885,43.750381],[1.000000,0.000000,0.000000,0.000000],[0,0,-1,0],[9E+09,9E+09,9E+09,9E+09,9E+09,9E+09]];
    CONST robtarget T4478:=[[45.249968,45.017502,44.250391],[1.000000,0.000000,0.000000,0.000000],[0,0,-1,0],[9E+09,9E+09,9E+09,9E+09,9E+09,9E+09]];
    CONST robtarget T4479:=[[45.249968,50.597754,44.250391],[1.000000,0.000000,0.000000,0.000000],[0,0,-1,0],[9E+09,9E+09,9E+09,9E+09,9E+09,9E+09]];
    CONST robtarget T4480:=[[45.249968,45.017502,44.250391],[1.000000,0.000000,0.000000,0.000000],[0,0,-1,0],[9E+09,9E+09,9E+09,9E+09,9E+09,9E+09]];
    CONST robtarget T4481:=[[45.249968,50.597754,44.250391],[1.000000,0.000000,0.000000,0.000000],[0,0,-1,0],[9E+09,9E+09,9E+09,9E+09,9E+09,9E+09]];
    CONST robtarget T4482:=[[46.749974,53.181615,44.250391],[1.000000,0.000000,0.000000,0.000000],[0,0,-1,0],[9E+09,9E+09,9E+09,9E+09,9E+09,9E+09]];
    CONST robtarget T4483:=[[46.749974,42.822104,44.250391],[1.000000,0.000000,0.000000,0.000000],[0,0,-1,0],[9E+09,9E+09,9E+09,9E+09,9E+09,9E+09]];
    CONST robtarget T4484:=[[48.249980,41.126777,44.250391],[1.000000,0.000000,0.000000,0.000000],[0,0,-1,0],[9E+09,9E+09,9E+09,9E+09,9E+09,9E+09]];
    CONST robtarget T4485:=[[48.249980,55.330319,44.250391],[1.000000,0.000000,0.000000,0.000000],[0,0,-1,0],[9E+09,9E+09,9E+09,9E+09,9E+09,9E+09]];
    CONST robtarget T4486:=[[49.749986,56.538540,44.250391],[1.000000,0.000000,0.000000,0.000000],[0,0,-1,0],[9E+09,9E+09,9E+09,9E+09,9E+09,9E+09]];
    CONST robtarget T4487:=[[49.749986,39.810365,44.250391],[1.000000,0.000000,0.000000,0.000000],[0,0,-1,0],[9E+09,9E+09,9E+09,9E+09,9E+09,9E+09]];
    CONST robtarget T4488:=[[51.249992,38.754058,44.250391],[1.000000,0.000000,0.000000,0.000000],[0,0,-1,0],[9E+09,9E+09,9E+09,9E+09,9E+09,9E+09]];
    CONST robtarget T4489:=[[51.249992,57.177358,44.250391],[1.000000,0.000000,0.000000,0.000000],[0,0,-1,0],[9E+09,9E+09,9E+09,9E+09,9E+09,9E+09]];
    CONST robtarget T4490:=[[52.749998,57.572565,44.250391],[1.000000,0.000000,0.000000,0.000000],[0,0,-1,0],[9E+09,9E+09,9E+09,9E+09,9E+09,9E+09]];
    CONST robtarget T4491:=[[52.749998,38.099748,44.250391],[1.000000,0.000000,0.000000,0.000000],[0,0,-1,0],[9E+09,9E+09,9E+09,9E+09,9E+09,9E+09]];
    CONST robtarget T4492:=[[54.250004,37.872769,44.250391],[1.000000,0.000000,0.000000,0.000000],[0,0,-1,0],[9E+09,9E+09,9E+09,9E+09,9E+09,9E+09]];
    CONST robtarget T4493:=[[54.250004,57.764626,44.250391],[1.000000,0.000000,0.000000,0.000000],[0,0,-1,0],[9E+09,9E+09,9E+09,9E+09,9E+09,9E+09]];
    CONST robtarget T4494:=[[55.750010,57.764626,44.250391],[1.000000,0.000000,0.000000,0.000000],[0,0,-1,0],[9E+09,9E+09,9E+09,9E+09,9E+09,9E+09]];
    CONST robtarget T4495:=[[55.750010,37.872765,44.250391],[1.000000,0.000000,0.000000,0.000000],[0,0,-1,0],[9E+09,9E+09,9E+09,9E+09,9E+09,9E+09]];
    CONST robtarget T4496:=[[57.250016,38.099748,44.250391],[1.000000,0.000000,0.000000,0.000000],[0,0,-1,0],[9E+09,9E+09,9E+09,9E+09,9E+09,9E+09]];
    CONST robtarget T4497:=[[57.250016,57.572565,44.250391],[1.000000,0.000000,0.000000,0.000000],[0,0,-1,0],[9E+09,9E+09,9E+09,9E+09,9E+09,9E+09]];
    CONST robtarget T4498:=[[58.750022,57.177358,44.250391],[1.000000,0.000000,0.000000,0.000000],[0,0,-1,0],[9E+09,9E+09,9E+09,9E+09,9E+09,9E+09]];
    CONST robtarget T4499:=[[58.750022,38.754067,44.250391],[1.000000,0.000000,0.000000,0.000000],[0,0,-1,0],[9E+09,9E+09,9E+09,9E+09,9E+09,9E+09]];
    CONST robtarget T4500:=[[60.250028,39.810363,44.250391],[1.000000,0.000000,0.000000,0.000000],[0,0,-1,0],[9E+09,9E+09,9E+09,9E+09,9E+09,9E+09]];
    CONST robtarget T4501:=[[60.250028,56.538539,44.250391],[1.000000,0.000000,0.000000,0.000000],[0,0,-1,0],[9E+09,9E+09,9E+09,9E+09,9E+09,9E+09]];
    CONST robtarget T4502:=[[61.750034,55.330318,44.250391],[1.000000,0.000000,0.000000,0.000000],[0,0,-1,0],[9E+09,9E+09,9E+09,9E+09,9E+09,9E+09]];
    CONST robtarget T4503:=[[61.750034,41.126774,44.250391],[1.000000,0.000000,0.000000,0.000000],[0,0,-1,0],[9E+09,9E+09,9E+09,9E+09,9E+09,9E+09]];
    CONST robtarget T4504:=[[63.250040,42.822105,44.250391],[1.000000,0.000000,0.000000,0.000000],[0,0,-1,0],[9E+09,9E+09,9E+09,9E+09,9E+09,9E+09]];
    CONST robtarget T4505:=[[63.250040,53.181616,44.250391],[1.000000,0.000000,0.000000,0.000000],[0,0,-1,0],[9E+09,9E+09,9E+09,9E+09,9E+09,9E+09]];
    CONST robtarget T4506:=[[64.750046,50.597754,44.250391],[1.000000,0.000000,0.000000,0.000000],[0,0,-1,0],[9E+09,9E+09,9E+09,9E+09,9E+09,9E+09]];
    CONST robtarget T4507:=[[64.750046,45.017502,44.250391],[1.000000,0.000000,0.000000,0.000000],[0,0,-1,0],[9E+09,9E+09,9E+09,9E+09,9E+09,9E+09]];
    CONST robtarget T4508:=[[64.750046,45.915180,44.750401],[1.000000,0.000000,0.000000,0.000000],[0,0,-1,0],[9E+09,9E+09,9E+09,9E+09,9E+09,9E+09]];
    CONST robtarget T4509:=[[64.750046,49.467067,44.750401],[1.000000,0.000000,0.000000,0.000000],[0,0,-1,0],[9E+09,9E+09,9E+09,9E+09,9E+09,9E+09]];
    CONST robtarget T4510:=[[64.750046,45.915180,44.750401],[1.000000,0.000000,0.000000,0.000000],[0,0,-1,0],[9E+09,9E+09,9E+09,9E+09,9E+09,9E+09]];
    CONST robtarget T4511:=[[64.750046,49.467067,44.750401],[1.000000,0.000000,0.000000,0.000000],[0,0,-1,0],[9E+09,9E+09,9E+09,9E+09,9E+09,9E+09]];
    CONST robtarget T4512:=[[63.250040,52.555408,44.750401],[1.000000,0.000000,0.000000,0.000000],[0,0,-1,0],[9E+09,9E+09,9E+09,9E+09,9E+09,9E+09]];
    CONST robtarget T4513:=[[63.250040,43.322621,44.750401],[1.000000,0.000000,0.000000,0.000000],[0,0,-1,0],[9E+09,9E+09,9E+09,9E+09,9E+09,9E+09]];
    CONST robtarget T4514:=[[61.750034,41.583658,44.750401],[1.000000,0.000000,0.000000,0.000000],[0,0,-1,0],[9E+09,9E+09,9E+09,9E+09,9E+09,9E+09]];
    CONST robtarget T4515:=[[61.750034,54.938196,44.750401],[1.000000,0.000000,0.000000,0.000000],[0,0,-1,0],[9E+09,9E+09,9E+09,9E+09,9E+09,9E+09]];
    CONST robtarget T4516:=[[60.250028,56.130700,44.750401],[1.000000,0.000000,0.000000,0.000000],[0,0,-1,0],[9E+09,9E+09,9E+09,9E+09,9E+09,9E+09]];
    CONST robtarget T4517:=[[60.250028,40.254421,44.750401],[1.000000,0.000000,0.000000,0.000000],[0,0,-1,0],[9E+09,9E+09,9E+09,9E+09,9E+09,9E+09]];
    CONST robtarget T4518:=[[58.750022,39.182871,44.750401],[1.000000,0.000000,0.000000,0.000000],[0,0,-1,0],[9E+09,9E+09,9E+09,9E+09,9E+09,9E+09]];
    CONST robtarget T4519:=[[58.750022,56.923810,44.750401],[1.000000,0.000000,0.000000,0.000000],[0,0,-1,0],[9E+09,9E+09,9E+09,9E+09,9E+09,9E+09]];
    CONST robtarget T4520:=[[57.250016,57.321988,44.750401],[1.000000,0.000000,0.000000,0.000000],[0,0,-1,0],[9E+09,9E+09,9E+09,9E+09,9E+09,9E+09]];
    CONST robtarget T4521:=[[57.250016,38.507590,44.750401],[1.000000,0.000000,0.000000,0.000000],[0,0,-1,0],[9E+09,9E+09,9E+09,9E+09,9E+09,9E+09]];
    CONST robtarget T4522:=[[55.750010,38.279565,44.750401],[1.000000,0.000000,0.000000,0.000000],[0,0,-1,0],[9E+09,9E+09,9E+09,9E+09,9E+09,9E+09]];
    CONST robtarget T4523:=[[55.750010,57.488298,44.750401],[1.000000,0.000000,0.000000,0.000000],[0,0,-1,0],[9E+09,9E+09,9E+09,9E+09,9E+09,9E+09]];
    CONST robtarget T4524:=[[54.250004,57.488298,44.750401],[1.000000,0.000000,0.000000,0.000000],[0,0,-1,0],[9E+09,9E+09,9E+09,9E+09,9E+09,9E+09]];
    CONST robtarget T4525:=[[54.250004,38.279568,44.750401],[1.000000,0.000000,0.000000,0.000000],[0,0,-1,0],[9E+09,9E+09,9E+09,9E+09,9E+09,9E+09]];
    CONST robtarget T4526:=[[52.749998,38.507590,44.750401],[1.000000,0.000000,0.000000,0.000000],[0,0,-1,0],[9E+09,9E+09,9E+09,9E+09,9E+09,9E+09]];
    CONST robtarget T4527:=[[52.749998,57.321988,44.750401],[1.000000,0.000000,0.000000,0.000000],[0,0,-1,0],[9E+09,9E+09,9E+09,9E+09,9E+09,9E+09]];
    CONST robtarget T4528:=[[51.249992,56.923810,44.750401],[1.000000,0.000000,0.000000,0.000000],[0,0,-1,0],[9E+09,9E+09,9E+09,9E+09,9E+09,9E+09]];
    CONST robtarget T4529:=[[51.249992,39.182862,44.750401],[1.000000,0.000000,0.000000,0.000000],[0,0,-1,0],[9E+09,9E+09,9E+09,9E+09,9E+09,9E+09]];
    CONST robtarget T4530:=[[49.749986,40.254426,44.750401],[1.000000,0.000000,0.000000,0.000000],[0,0,-1,0],[9E+09,9E+09,9E+09,9E+09,9E+09,9E+09]];
    CONST robtarget T4531:=[[49.749986,56.130701,44.750401],[1.000000,0.000000,0.000000,0.000000],[0,0,-1,0],[9E+09,9E+09,9E+09,9E+09,9E+09,9E+09]];
    CONST robtarget T4532:=[[48.249980,54.938197,44.750401],[1.000000,0.000000,0.000000,0.000000],[0,0,-1,0],[9E+09,9E+09,9E+09,9E+09,9E+09,9E+09]];
    CONST robtarget T4533:=[[48.249980,41.583659,44.750401],[1.000000,0.000000,0.000000,0.000000],[0,0,-1,0],[9E+09,9E+09,9E+09,9E+09,9E+09,9E+09]];
    CONST robtarget T4534:=[[46.749974,43.322620,44.750401],[1.000000,0.000000,0.000000,0.000000],[0,0,-1,0],[9E+09,9E+09,9E+09,9E+09,9E+09,9E+09]];
    CONST robtarget T4535:=[[46.749974,52.555408,44.750401],[1.000000,0.000000,0.000000,0.000000],[0,0,-1,0],[9E+09,9E+09,9E+09,9E+09,9E+09,9E+09]];
    CONST robtarget T4536:=[[45.249968,49.467067,44.750401],[1.000000,0.000000,0.000000,0.000000],[0,0,-1,0],[9E+09,9E+09,9E+09,9E+09,9E+09,9E+09]];
    CONST robtarget T4537:=[[45.249968,45.915179,44.750401],[1.000000,0.000000,0.000000,0.000000],[0,0,-1,0],[9E+09,9E+09,9E+09,9E+09,9E+09,9E+09]];
    CONST robtarget T4538:=[[45.999971,45.081002,45.250411],[1.000000,0.000000,0.000000,0.000000],[0,0,-1,0],[9E+09,9E+09,9E+09,9E+09,9E+09,9E+09]];
    CONST robtarget T4539:=[[45.999971,50.147179,45.250411],[1.000000,0.000000,0.000000,0.000000],[0,0,-1,0],[9E+09,9E+09,9E+09,9E+09,9E+09,9E+09]];
    CONST robtarget T4540:=[[45.999971,45.081002,45.250411],[1.000000,0.000000,0.000000,0.000000],[0,0,-1,0],[9E+09,9E+09,9E+09,9E+09,9E+09,9E+09]];
    CONST robtarget T4541:=[[45.999971,50.147179,45.250411],[1.000000,0.000000,0.000000,0.000000],[0,0,-1,0],[9E+09,9E+09,9E+09,9E+09,9E+09,9E+09]];
    CONST robtarget T4542:=[[47.499977,53.202434,45.250411],[1.000000,0.000000,0.000000,0.000000],[0,0,-1,0],[9E+09,9E+09,9E+09,9E+09,9E+09,9E+09]];
    CONST robtarget T4543:=[[47.499977,42.991934,45.250411],[1.000000,0.000000,0.000000,0.000000],[0,0,-1,0],[9E+09,9E+09,9E+09,9E+09,9E+09,9E+09]];
    CONST robtarget T4544:=[[48.999983,41.451984,45.250411],[1.000000,0.000000,0.000000,0.000000],[0,0,-1,0],[9E+09,9E+09,9E+09,9E+09,9E+09,9E+09]];
    CONST robtarget T4545:=[[48.999983,55.108248,45.250411],[1.000000,0.000000,0.000000,0.000000],[0,0,-1,0],[9E+09,9E+09,9E+09,9E+09,9E+09,9E+09]];
    CONST robtarget T4546:=[[50.499989,56.293087,45.250411],[1.000000,0.000000,0.000000,0.000000],[0,0,-1,0],[9E+09,9E+09,9E+09,9E+09,9E+09,9E+09]];
    CONST robtarget T4547:=[[50.499989,40.106610,45.250411],[1.000000,0.000000,0.000000,0.000000],[0,0,-1,0],[9E+09,9E+09,9E+09,9E+09,9E+09,9E+09]];
    CONST robtarget T4548:=[[51.999995,39.241227,45.250411],[1.000000,0.000000,0.000000,0.000000],[0,0,-1,0],[9E+09,9E+09,9E+09,9E+09,9E+09,9E+09]];
    CONST robtarget T4549:=[[51.999995,56.906208,45.250411],[1.000000,0.000000,0.000000,0.000000],[0,0,-1,0],[9E+09,9E+09,9E+09,9E+09,9E+09,9E+09]];
    CONST robtarget T4550:=[[53.500001,57.171239,45.250411],[1.000000,0.000000,0.000000,0.000000],[0,0,-1,0],[9E+09,9E+09,9E+09,9E+09,9E+09,9E+09]];
    CONST robtarget T4551:=[[53.500001,38.765047,45.250411],[1.000000,0.000000,0.000000,0.000000],[0,0,-1,0],[9E+09,9E+09,9E+09,9E+09,9E+09,9E+09]];
    CONST robtarget T4552:=[[55.000007,38.686654,45.250411],[1.000000,0.000000,0.000000,0.000000],[0,0,-1,0],[9E+09,9E+09,9E+09,9E+09,9E+09,9E+09]];
    CONST robtarget T4553:=[[55.000007,57.248613,45.250411],[1.000000,0.000000,0.000000,0.000000],[0,0,-1,0],[9E+09,9E+09,9E+09,9E+09,9E+09,9E+09]];
    CONST robtarget T4554:=[[56.500013,57.171239,45.250411],[1.000000,0.000000,0.000000,0.000000],[0,0,-1,0],[9E+09,9E+09,9E+09,9E+09,9E+09,9E+09]];
    CONST robtarget T4555:=[[56.500013,38.765047,45.250411],[1.000000,0.000000,0.000000,0.000000],[0,0,-1,0],[9E+09,9E+09,9E+09,9E+09,9E+09,9E+09]];
    CONST robtarget T4556:=[[58.000019,39.241230,45.250411],[1.000000,0.000000,0.000000,0.000000],[0,0,-1,0],[9E+09,9E+09,9E+09,9E+09,9E+09,9E+09]];
    CONST robtarget T4557:=[[58.000019,56.906207,45.250411],[1.000000,0.000000,0.000000,0.000000],[0,0,-1,0],[9E+09,9E+09,9E+09,9E+09,9E+09,9E+09]];
    CONST robtarget T4558:=[[59.500025,56.293086,45.250411],[1.000000,0.000000,0.000000,0.000000],[0,0,-1,0],[9E+09,9E+09,9E+09,9E+09,9E+09,9E+09]];
    CONST robtarget T4559:=[[59.500025,40.106611,45.250411],[1.000000,0.000000,0.000000,0.000000],[0,0,-1,0],[9E+09,9E+09,9E+09,9E+09,9E+09,9E+09]];
    CONST robtarget T4560:=[[61.000031,41.451983,45.250411],[1.000000,0.000000,0.000000,0.000000],[0,0,-1,0],[9E+09,9E+09,9E+09,9E+09,9E+09,9E+09]];
    CONST robtarget T4561:=[[61.000031,55.108247,45.250411],[1.000000,0.000000,0.000000,0.000000],[0,0,-1,0],[9E+09,9E+09,9E+09,9E+09,9E+09,9E+09]];
    CONST robtarget T4562:=[[62.500037,53.202433,45.250411],[1.000000,0.000000,0.000000,0.000000],[0,0,-1,0],[9E+09,9E+09,9E+09,9E+09,9E+09,9E+09]];
    CONST robtarget T4563:=[[62.500037,42.991935,45.250411],[1.000000,0.000000,0.000000,0.000000],[0,0,-1,0],[9E+09,9E+09,9E+09,9E+09,9E+09,9E+09]];
    CONST robtarget T4564:=[[64.000043,45.081002,45.250411],[1.000000,0.000000,0.000000,0.000000],[0,0,-1,0],[9E+09,9E+09,9E+09,9E+09,9E+09,9E+09]];
    CONST robtarget T4565:=[[64.000043,50.147178,45.250411],[1.000000,0.000000,0.000000,0.000000],[0,0,-1,0],[9E+09,9E+09,9E+09,9E+09,9E+09,9E+09]];
    CONST robtarget T4566:=[[63.250040,44.678958,45.750421],[1.000000,0.000000,0.000000,0.000000],[0,0,-1,0],[9E+09,9E+09,9E+09,9E+09,9E+09,9E+09]];
    CONST robtarget T4567:=[[63.250040,50.827290,45.750421],[1.000000,0.000000,0.000000,0.000000],[0,0,-1,0],[9E+09,9E+09,9E+09,9E+09,9E+09,9E+09]];
    CONST robtarget T4568:=[[63.250040,44.678958,45.750421],[1.000000,0.000000,0.000000,0.000000],[0,0,-1,0],[9E+09,9E+09,9E+09,9E+09,9E+09,9E+09]];
    CONST robtarget T4569:=[[63.250040,50.827290,45.750421],[1.000000,0.000000,0.000000,0.000000],[0,0,-1,0],[9E+09,9E+09,9E+09,9E+09,9E+09,9E+09]];
    CONST robtarget T4570:=[[61.750034,53.574940,45.750421],[1.000000,0.000000,0.000000,0.000000],[0,0,-1,0],[9E+09,9E+09,9E+09,9E+09,9E+09,9E+09]];
    CONST robtarget T4571:=[[61.750034,42.712080,45.750421],[1.000000,0.000000,0.000000,0.000000],[0,0,-1,0],[9E+09,9E+09,9E+09,9E+09,9E+09,9E+09]];
    CONST robtarget T4572:=[[60.250028,41.320308,45.750421],[1.000000,0.000000,0.000000,0.000000],[0,0,-1,0],[9E+09,9E+09,9E+09,9E+09,9E+09,9E+09]];
    CONST robtarget T4573:=[[60.250028,55.315024,45.750421],[1.000000,0.000000,0.000000,0.000000],[0,0,-1,0],[9E+09,9E+09,9E+09,9E+09,9E+09,9E+09]];
    CONST robtarget T4574:=[[58.750022,56.286882,45.750421],[1.000000,0.000000,0.000000,0.000000],[0,0,-1,0],[9E+09,9E+09,9E+09,9E+09,9E+09,9E+09]];
    CONST robtarget T4575:=[[58.750022,40.149986,45.750421],[1.000000,0.000000,0.000000,0.000000],[0,0,-1,0],[9E+09,9E+09,9E+09,9E+09,9E+09,9E+09]];
    CONST robtarget T4576:=[[57.250016,39.444137,45.750421],[1.000000,0.000000,0.000000,0.000000],[0,0,-1,0],[9E+09,9E+09,9E+09,9E+09,9E+09,9E+09]];
    CONST robtarget T4577:=[[57.250016,56.779012,45.750421],[1.000000,0.000000,0.000000,0.000000],[0,0,-1,0],[9E+09,9E+09,9E+09,9E+09,9E+09,9E+09]];
    CONST robtarget T4578:=[[55.750010,56.926744,45.750421],[1.000000,0.000000,0.000000,0.000000],[0,0,-1,0],[9E+09,9E+09,9E+09,9E+09,9E+09,9E+09]];
    CONST robtarget T4579:=[[55.750010,39.185727,45.750421],[1.000000,0.000000,0.000000,0.000000],[0,0,-1,0],[9E+09,9E+09,9E+09,9E+09,9E+09,9E+09]];
    CONST robtarget T4580:=[[54.250004,39.185727,45.750421],[1.000000,0.000000,0.000000,0.000000],[0,0,-1,0],[9E+09,9E+09,9E+09,9E+09,9E+09,9E+09]];
    CONST robtarget T4581:=[[54.250004,56.926744,45.750421],[1.000000,0.000000,0.000000,0.000000],[0,0,-1,0],[9E+09,9E+09,9E+09,9E+09,9E+09,9E+09]];
    CONST robtarget T4582:=[[52.749998,56.779012,45.750421],[1.000000,0.000000,0.000000,0.000000],[0,0,-1,0],[9E+09,9E+09,9E+09,9E+09,9E+09,9E+09]];
    CONST robtarget T4583:=[[52.749998,39.444137,45.750421],[1.000000,0.000000,0.000000,0.000000],[0,0,-1,0],[9E+09,9E+09,9E+09,9E+09,9E+09,9E+09]];
    CONST robtarget T4584:=[[51.249992,40.149986,45.750421],[1.000000,0.000000,0.000000,0.000000],[0,0,-1,0],[9E+09,9E+09,9E+09,9E+09,9E+09,9E+09]];
    CONST robtarget T4585:=[[51.249992,56.286883,45.750421],[1.000000,0.000000,0.000000,0.000000],[0,0,-1,0],[9E+09,9E+09,9E+09,9E+09,9E+09,9E+09]];
    CONST robtarget T4586:=[[49.749986,55.315025,45.750421],[1.000000,0.000000,0.000000,0.000000],[0,0,-1,0],[9E+09,9E+09,9E+09,9E+09,9E+09,9E+09]];
    CONST robtarget T4587:=[[49.749986,41.320309,45.750421],[1.000000,0.000000,0.000000,0.000000],[0,0,-1,0],[9E+09,9E+09,9E+09,9E+09,9E+09,9E+09]];
    CONST robtarget T4588:=[[48.249980,42.712079,45.750421],[1.000000,0.000000,0.000000,0.000000],[0,0,-1,0],[9E+09,9E+09,9E+09,9E+09,9E+09,9E+09]];
    CONST robtarget T4589:=[[48.249980,53.574941,45.750421],[1.000000,0.000000,0.000000,0.000000],[0,0,-1,0],[9E+09,9E+09,9E+09,9E+09,9E+09,9E+09]];
    CONST robtarget T4590:=[[46.749974,50.827291,45.750421],[1.000000,0.000000,0.000000,0.000000],[0,0,-1,0],[9E+09,9E+09,9E+09,9E+09,9E+09,9E+09]];
    CONST robtarget T4591:=[[46.749974,44.678957,45.750421],[1.000000,0.000000,0.000000,0.000000],[0,0,-1,0],[9E+09,9E+09,9E+09,9E+09,9E+09,9E+09]];
    CONST robtarget T4592:=[[47.499977,44.324900,46.250431],[1.000000,0.000000,0.000000,0.000000],[0,0,-1,0],[9E+09,9E+09,9E+09,9E+09,9E+09,9E+09]];
    CONST robtarget T4593:=[[47.499977,50.981029,46.250431],[1.000000,0.000000,0.000000,0.000000],[0,0,-1,0],[9E+09,9E+09,9E+09,9E+09,9E+09,9E+09]];
    CONST robtarget T4594:=[[47.499977,44.324900,46.250431],[1.000000,0.000000,0.000000,0.000000],[0,0,-1,0],[9E+09,9E+09,9E+09,9E+09,9E+09,9E+09]];
    CONST robtarget T4595:=[[47.499977,50.981029,46.250431],[1.000000,0.000000,0.000000,0.000000],[0,0,-1,0],[9E+09,9E+09,9E+09,9E+09,9E+09,9E+09]];
    CONST robtarget T4596:=[[48.999983,53.944662,46.250431],[1.000000,0.000000,0.000000,0.000000],[0,0,-1,0],[9E+09,9E+09,9E+09,9E+09,9E+09,9E+09]];
    CONST robtarget T4597:=[[48.999983,42.594878,46.250431],[1.000000,0.000000,0.000000,0.000000],[0,0,-1,0],[9E+09,9E+09,9E+09,9E+09,9E+09,9E+09]];
    CONST robtarget T4598:=[[50.499989,41.257013,46.250431],[1.000000,0.000000,0.000000,0.000000],[0,0,-1,0],[9E+09,9E+09,9E+09,9E+09,9E+09,9E+09]];
    CONST robtarget T4599:=[[50.499989,55.360473,46.250431],[1.000000,0.000000,0.000000,0.000000],[0,0,-1,0],[9E+09,9E+09,9E+09,9E+09,9E+09,9E+09]];
    CONST robtarget T4600:=[[51.999995,56.246037,46.250431],[1.000000,0.000000,0.000000,0.000000],[0,0,-1,0],[9E+09,9E+09,9E+09,9E+09,9E+09,9E+09]];
    CONST robtarget T4601:=[[51.999995,40.226734,46.250431],[1.000000,0.000000,0.000000,0.000000],[0,0,-1,0],[9E+09,9E+09,9E+09,9E+09,9E+09,9E+09]];
    CONST robtarget T4602:=[[53.500001,39.765081,46.250431],[1.000000,0.000000,0.000000,0.000000],[0,0,-1,0],[9E+09,9E+09,9E+09,9E+09,9E+09,9E+09]];
    CONST robtarget T4603:=[[53.500001,56.623917,46.250431],[1.000000,0.000000,0.000000,0.000000],[0,0,-1,0],[9E+09,9E+09,9E+09,9E+09,9E+09,9E+09]];
    CONST robtarget T4604:=[[55.000007,56.678178,46.250431],[1.000000,0.000000,0.000000,0.000000],[0,0,-1,0],[9E+09,9E+09,9E+09,9E+09,9E+09,9E+09]];
    CONST robtarget T4605:=[[55.000007,39.688141,46.250431],[1.000000,0.000000,0.000000,0.000000],[0,0,-1,0],[9E+09,9E+09,9E+09,9E+09,9E+09,9E+09]];
    CONST robtarget T4606:=[[56.500013,39.765082,46.250431],[1.000000,0.000000,0.000000,0.000000],[0,0,-1,0],[9E+09,9E+09,9E+09,9E+09,9E+09,9E+09]];
    CONST robtarget T4607:=[[56.500013,56.623917,46.250431],[1.000000,0.000000,0.000000,0.000000],[0,0,-1,0],[9E+09,9E+09,9E+09,9E+09,9E+09,9E+09]];
    CONST robtarget T4608:=[[58.000019,56.246037,46.250431],[1.000000,0.000000,0.000000,0.000000],[0,0,-1,0],[9E+09,9E+09,9E+09,9E+09,9E+09,9E+09]];
    CONST robtarget T4609:=[[58.000019,40.226734,46.250431],[1.000000,0.000000,0.000000,0.000000],[0,0,-1,0],[9E+09,9E+09,9E+09,9E+09,9E+09,9E+09]];
    CONST robtarget T4610:=[[59.500025,41.257013,46.250431],[1.000000,0.000000,0.000000,0.000000],[0,0,-1,0],[9E+09,9E+09,9E+09,9E+09,9E+09,9E+09]];
    CONST robtarget T4611:=[[59.500025,55.360472,46.250431],[1.000000,0.000000,0.000000,0.000000],[0,0,-1,0],[9E+09,9E+09,9E+09,9E+09,9E+09,9E+09]];
    CONST robtarget T4612:=[[61.000031,53.944660,46.250431],[1.000000,0.000000,0.000000,0.000000],[0,0,-1,0],[9E+09,9E+09,9E+09,9E+09,9E+09,9E+09]];
    CONST robtarget T4613:=[[61.000031,42.594877,46.250431],[1.000000,0.000000,0.000000,0.000000],[0,0,-1,0],[9E+09,9E+09,9E+09,9E+09,9E+09,9E+09]];
    CONST robtarget T4614:=[[62.500037,44.324901,46.250431],[1.000000,0.000000,0.000000,0.000000],[0,0,-1,0],[9E+09,9E+09,9E+09,9E+09,9E+09,9E+09]];
    CONST robtarget T4615:=[[62.500037,50.981028,46.250431],[1.000000,0.000000,0.000000,0.000000],[0,0,-1,0],[9E+09,9E+09,9E+09,9E+09,9E+09,9E+09]];
    CONST robtarget T4616:=[[62.500038,45.344222,46.750441],[1.000000,0.000000,0.000000,0.000000],[0,0,-1,0],[9E+09,9E+09,9E+09,9E+09,9E+09,9E+09]];
    CONST robtarget T4617:=[[62.500038,49.423553,46.750441],[1.000000,0.000000,0.000000,0.000000],[0,0,-1,0],[9E+09,9E+09,9E+09,9E+09,9E+09,9E+09]];
    CONST robtarget T4618:=[[62.500038,45.344222,46.750441],[1.000000,0.000000,0.000000,0.000000],[0,0,-1,0],[9E+09,9E+09,9E+09,9E+09,9E+09,9E+09]];
    CONST robtarget T4619:=[[62.500038,49.423553,46.750441],[1.000000,0.000000,0.000000,0.000000],[0,0,-1,0],[9E+09,9E+09,9E+09,9E+09,9E+09,9E+09]];
    CONST robtarget T4620:=[[61.000032,52.866144,46.750441],[1.000000,0.000000,0.000000,0.000000],[0,0,-1,0],[9E+09,9E+09,9E+09,9E+09,9E+09,9E+09]];
    CONST robtarget T4621:=[[61.000032,43.281661,46.750441],[1.000000,0.000000,0.000000,0.000000],[0,0,-1,0],[9E+09,9E+09,9E+09,9E+09,9E+09,9E+09]];
    CONST robtarget T4622:=[[59.500026,41.932595,46.750441],[1.000000,0.000000,0.000000,0.000000],[0,0,-1,0],[9E+09,9E+09,9E+09,9E+09,9E+09,9E+09]];
    CONST robtarget T4623:=[[59.500026,54.896374,46.750441],[1.000000,0.000000,0.000000,0.000000],[0,0,-1,0],[9E+09,9E+09,9E+09,9E+09,9E+09,9E+09]];
    CONST robtarget T4624:=[[58.000020,55.737157,46.750441],[1.000000,0.000000,0.000000,0.000000],[0,0,-1,0],[9E+09,9E+09,9E+09,9E+09,9E+09,9E+09]];
    CONST robtarget T4625:=[[58.000020,40.818327,46.750441],[1.000000,0.000000,0.000000,0.000000],[0,0,-1,0],[9E+09,9E+09,9E+09,9E+09,9E+09,9E+09]];
    CONST robtarget T4626:=[[56.500014,40.318287,46.750441],[1.000000,0.000000,0.000000,0.000000],[0,0,-1,0],[9E+09,9E+09,9E+09,9E+09,9E+09,9E+09]];
    CONST robtarget T4627:=[[56.500014,56.175908,46.750441],[1.000000,0.000000,0.000000,0.000000],[0,0,-1,0],[9E+09,9E+09,9E+09,9E+09,9E+09,9E+09]];
    CONST robtarget T4628:=[[55.000008,56.181245,46.750441],[1.000000,0.000000,0.000000,0.000000],[0,0,-1,0],[9E+09,9E+09,9E+09,9E+09,9E+09,9E+09]];
    CONST robtarget T4629:=[[55.000008,40.239786,46.750441],[1.000000,0.000000,0.000000,0.000000],[0,0,-1,0],[9E+09,9E+09,9E+09,9E+09,9E+09,9E+09]];
    CONST robtarget T4630:=[[53.500002,40.318287,46.750441],[1.000000,0.000000,0.000000,0.000000],[0,0,-1,0],[9E+09,9E+09,9E+09,9E+09,9E+09,9E+09]];
    CONST robtarget T4631:=[[53.500002,56.175908,46.750441],[1.000000,0.000000,0.000000,0.000000],[0,0,-1,0],[9E+09,9E+09,9E+09,9E+09,9E+09,9E+09]];
    CONST robtarget T4632:=[[51.999996,55.737157,46.750441],[1.000000,0.000000,0.000000,0.000000],[0,0,-1,0],[9E+09,9E+09,9E+09,9E+09,9E+09,9E+09]];
    CONST robtarget T4633:=[[51.999996,40.818327,46.750441],[1.000000,0.000000,0.000000,0.000000],[0,0,-1,0],[9E+09,9E+09,9E+09,9E+09,9E+09,9E+09]];
    CONST robtarget T4634:=[[50.499990,41.932593,46.750441],[1.000000,0.000000,0.000000,0.000000],[0,0,-1,0],[9E+09,9E+09,9E+09,9E+09,9E+09,9E+09]];
    CONST robtarget T4635:=[[50.499990,54.896375,46.750441],[1.000000,0.000000,0.000000,0.000000],[0,0,-1,0],[9E+09,9E+09,9E+09,9E+09,9E+09,9E+09]];
    CONST robtarget T4636:=[[48.999984,52.866146,46.750441],[1.000000,0.000000,0.000000,0.000000],[0,0,-1,0],[9E+09,9E+09,9E+09,9E+09,9E+09,9E+09]];
    CONST robtarget T4637:=[[48.999984,43.281670,46.750441],[1.000000,0.000000,0.000000,0.000000],[0,0,-1,0],[9E+09,9E+09,9E+09,9E+09,9E+09,9E+09]];
    CONST robtarget T4638:=[[47.499978,45.344219,46.750441],[1.000000,0.000000,0.000000,0.000000],[0,0,-1,0],[9E+09,9E+09,9E+09,9E+09,9E+09,9E+09]];
    CONST robtarget T4639:=[[47.499978,49.423554,46.750441],[1.000000,0.000000,0.000000,0.000000],[0,0,-1,0],[9E+09,9E+09,9E+09,9E+09,9E+09,9E+09]];
    CONST robtarget T4640:=[[48.249980,45.409553,47.250451],[1.000000,0.000000,0.000000,0.000000],[0,0,-1,0],[9E+09,9E+09,9E+09,9E+09,9E+09,9E+09]];
    CONST robtarget T4641:=[[48.249980,49.501457,47.250451],[1.000000,0.000000,0.000000,0.000000],[0,0,-1,0],[9E+09,9E+09,9E+09,9E+09,9E+09,9E+09]];
    CONST robtarget T4642:=[[48.249980,45.409553,47.250451],[1.000000,0.000000,0.000000,0.000000],[0,0,-1,0],[9E+09,9E+09,9E+09,9E+09,9E+09,9E+09]];
    CONST robtarget T4643:=[[48.249980,49.501457,47.250451],[1.000000,0.000000,0.000000,0.000000],[0,0,-1,0],[9E+09,9E+09,9E+09,9E+09,9E+09,9E+09]];
    CONST robtarget T4644:=[[49.749986,52.957566,47.250451],[1.000000,0.000000,0.000000,0.000000],[0,0,-1,0],[9E+09,9E+09,9E+09,9E+09,9E+09,9E+09]];
    CONST robtarget T4645:=[[49.749986,43.227394,47.250451],[1.000000,0.000000,0.000000,0.000000],[0,0,-1,0],[9E+09,9E+09,9E+09,9E+09,9E+09,9E+09]];
    CONST robtarget T4646:=[[51.249992,42.041259,47.250451],[1.000000,0.000000,0.000000,0.000000],[0,0,-1,0],[9E+09,9E+09,9E+09,9E+09,9E+09,9E+09]];
    CONST robtarget T4647:=[[51.249992,54.893129,47.250451],[1.000000,0.000000,0.000000,0.000000],[0,0,-1,0],[9E+09,9E+09,9E+09,9E+09,9E+09,9E+09]];
    CONST robtarget T4648:=[[52.749998,55.421142,47.250451],[1.000000,0.000000,0.000000,0.000000],[0,0,-1,0],[9E+09,9E+09,9E+09,9E+09,9E+09,9E+09]];
    CONST robtarget T4649:=[[52.749998,41.176419,47.250451],[1.000000,0.000000,0.000000,0.000000],[0,0,-1,0],[9E+09,9E+09,9E+09,9E+09,9E+09,9E+09]];
    CONST robtarget T4650:=[[54.250004,40.892656,47.250451],[1.000000,0.000000,0.000000,0.000000],[0,0,-1,0],[9E+09,9E+09,9E+09,9E+09,9E+09,9E+09]];
    CONST robtarget T4651:=[[54.250004,55.632273,47.250451],[1.000000,0.000000,0.000000,0.000000],[0,0,-1,0],[9E+09,9E+09,9E+09,9E+09,9E+09,9E+09]];
    CONST robtarget T4652:=[[55.750010,55.632273,47.250451],[1.000000,0.000000,0.000000,0.000000],[0,0,-1,0],[9E+09,9E+09,9E+09,9E+09,9E+09,9E+09]];
    CONST robtarget T4653:=[[55.750010,40.892656,47.250451],[1.000000,0.000000,0.000000,0.000000],[0,0,-1,0],[9E+09,9E+09,9E+09,9E+09,9E+09,9E+09]];
    CONST robtarget T4654:=[[57.250016,41.176420,47.250451],[1.000000,0.000000,0.000000,0.000000],[0,0,-1,0],[9E+09,9E+09,9E+09,9E+09,9E+09,9E+09]];
    CONST robtarget T4655:=[[57.250016,55.421141,47.250451],[1.000000,0.000000,0.000000,0.000000],[0,0,-1,0],[9E+09,9E+09,9E+09,9E+09,9E+09,9E+09]];
    CONST robtarget T4656:=[[58.750022,54.893128,47.250451],[1.000000,0.000000,0.000000,0.000000],[0,0,-1,0],[9E+09,9E+09,9E+09,9E+09,9E+09,9E+09]];
    CONST robtarget T4657:=[[58.750022,42.041263,47.250451],[1.000000,0.000000,0.000000,0.000000],[0,0,-1,0],[9E+09,9E+09,9E+09,9E+09,9E+09,9E+09]];
    CONST robtarget T4658:=[[60.250028,43.227377,47.250451],[1.000000,0.000000,0.000000,0.000000],[0,0,-1,0],[9E+09,9E+09,9E+09,9E+09,9E+09,9E+09]];
    CONST robtarget T4659:=[[60.250028,52.957565,47.250451],[1.000000,0.000000,0.000000,0.000000],[0,0,-1,0],[9E+09,9E+09,9E+09,9E+09,9E+09,9E+09]];
    CONST robtarget T4660:=[[61.750034,49.501456,47.250451],[1.000000,0.000000,0.000000,0.000000],[0,0,-1,0],[9E+09,9E+09,9E+09,9E+09,9E+09,9E+09]];
    CONST robtarget T4661:=[[61.750034,45.409555,47.250451],[1.000000,0.000000,0.000000,0.000000],[0,0,-1,0],[9E+09,9E+09,9E+09,9E+09,9E+09,9E+09]];
    CONST robtarget T4662:=[[61.000031,45.456231,47.750461],[1.000000,0.000000,0.000000,0.000000],[0,0,-1,0],[9E+09,9E+09,9E+09,9E+09,9E+09,9E+09]];
    CONST robtarget T4663:=[[61.000031,49.796809,47.750461],[1.000000,0.000000,0.000000,0.000000],[0,0,-1,0],[9E+09,9E+09,9E+09,9E+09,9E+09,9E+09]];
    CONST robtarget T4664:=[[61.000031,45.456231,47.750461],[1.000000,0.000000,0.000000,0.000000],[0,0,-1,0],[9E+09,9E+09,9E+09,9E+09,9E+09,9E+09]];
    CONST robtarget T4665:=[[61.000031,49.796809,47.750461],[1.000000,0.000000,0.000000,0.000000],[0,0,-1,0],[9E+09,9E+09,9E+09,9E+09,9E+09,9E+09]];
    CONST robtarget T4666:=[[59.500025,52.820343,47.750461],[1.000000,0.000000,0.000000,0.000000],[0,0,-1,0],[9E+09,9E+09,9E+09,9E+09,9E+09,9E+09]];
    CONST robtarget T4667:=[[59.500025,43.446546,47.750461],[1.000000,0.000000,0.000000,0.000000],[0,0,-1,0],[9E+09,9E+09,9E+09,9E+09,9E+09,9E+09]];
    CONST robtarget T4668:=[[58.000019,42.194975,47.750461],[1.000000,0.000000,0.000000,0.000000],[0,0,-1,0],[9E+09,9E+09,9E+09,9E+09,9E+09,9E+09]];
    CONST robtarget T4669:=[[58.000019,54.716494,47.750461],[1.000000,0.000000,0.000000,0.000000],[0,0,-1,0],[9E+09,9E+09,9E+09,9E+09,9E+09,9E+09]];
    CONST robtarget T4670:=[[56.500013,55.081629,47.750461],[1.000000,0.000000,0.000000,0.000000],[0,0,-1,0],[9E+09,9E+09,9E+09,9E+09,9E+09,9E+09]];
    CONST robtarget T4671:=[[56.500013,41.584973,47.750461],[1.000000,0.000000,0.000000,0.000000],[0,0,-1,0],[9E+09,9E+09,9E+09,9E+09,9E+09,9E+09]];
    CONST robtarget T4672:=[[55.000007,41.507640,47.750461],[1.000000,0.000000,0.000000,0.000000],[0,0,-1,0],[9E+09,9E+09,9E+09,9E+09,9E+09,9E+09]];
    CONST robtarget T4673:=[[55.000007,55.073441,47.750461],[1.000000,0.000000,0.000000,0.000000],[0,0,-1,0],[9E+09,9E+09,9E+09,9E+09,9E+09,9E+09]];
    CONST robtarget T4674:=[[53.500001,55.081629,47.750461],[1.000000,0.000000,0.000000,0.000000],[0,0,-1,0],[9E+09,9E+09,9E+09,9E+09,9E+09,9E+09]];
    CONST robtarget T4675:=[[53.500001,41.584971,47.750461],[1.000000,0.000000,0.000000,0.000000],[0,0,-1,0],[9E+09,9E+09,9E+09,9E+09,9E+09,9E+09]];
    CONST robtarget T4676:=[[51.999995,42.194969,47.750461],[1.000000,0.000000,0.000000,0.000000],[0,0,-1,0],[9E+09,9E+09,9E+09,9E+09,9E+09,9E+09]];
    CONST robtarget T4677:=[[51.999995,54.716494,47.750461],[1.000000,0.000000,0.000000,0.000000],[0,0,-1,0],[9E+09,9E+09,9E+09,9E+09,9E+09,9E+09]];
    CONST robtarget T4678:=[[50.499989,52.820344,47.750461],[1.000000,0.000000,0.000000,0.000000],[0,0,-1,0],[9E+09,9E+09,9E+09,9E+09,9E+09,9E+09]];
    CONST robtarget T4679:=[[50.499989,43.446547,47.750461],[1.000000,0.000000,0.000000,0.000000],[0,0,-1,0],[9E+09,9E+09,9E+09,9E+09,9E+09,9E+09]];
    CONST robtarget T4680:=[[48.999983,45.456231,47.750461],[1.000000,0.000000,0.000000,0.000000],[0,0,-1,0],[9E+09,9E+09,9E+09,9E+09,9E+09,9E+09]];
    CONST robtarget T4681:=[[48.999983,49.796810,47.750461],[1.000000,0.000000,0.000000,0.000000],[0,0,-1,0],[9E+09,9E+09,9E+09,9E+09,9E+09,9E+09]];
    CONST robtarget T4682:=[[49.749986,45.646615,48.250471],[1.000000,0.000000,0.000000,0.000000],[0,0,-1,0],[9E+09,9E+09,9E+09,9E+09,9E+09,9E+09]];
    CONST robtarget T4683:=[[49.749986,49.742584,48.250471],[1.000000,0.000000,0.000000,0.000000],[0,0,-1,0],[9E+09,9E+09,9E+09,9E+09,9E+09,9E+09]];
    CONST robtarget T4684:=[[49.749986,45.646615,48.250471],[1.000000,0.000000,0.000000,0.000000],[0,0,-1,0],[9E+09,9E+09,9E+09,9E+09,9E+09,9E+09]];
    CONST robtarget T4685:=[[49.749986,49.742584,48.250471],[1.000000,0.000000,0.000000,0.000000],[0,0,-1,0],[9E+09,9E+09,9E+09,9E+09,9E+09,9E+09]];
    CONST robtarget T4686:=[[51.249992,52.734295,48.250471],[1.000000,0.000000,0.000000,0.000000],[0,0,-1,0],[9E+09,9E+09,9E+09,9E+09,9E+09,9E+09]];
    CONST robtarget T4687:=[[51.249992,43.675927,48.250471],[1.000000,0.000000,0.000000,0.000000],[0,0,-1,0],[9E+09,9E+09,9E+09,9E+09,9E+09,9E+09]];
    CONST robtarget T4688:=[[52.749998,42.694176,48.250471],[1.000000,0.000000,0.000000,0.000000],[0,0,-1,0],[9E+09,9E+09,9E+09,9E+09,9E+09,9E+09]];
    CONST robtarget T4689:=[[52.749998,53.932207,48.250471],[1.000000,0.000000,0.000000,0.000000],[0,0,-1,0],[9E+09,9E+09,9E+09,9E+09,9E+09,9E+09]];
    CONST robtarget T4690:=[[54.250004,54.272228,48.250471],[1.000000,0.000000,0.000000,0.000000],[0,0,-1,0],[9E+09,9E+09,9E+09,9E+09,9E+09,9E+09]];
    CONST robtarget T4691:=[[54.250004,42.356439,48.250471],[1.000000,0.000000,0.000000,0.000000],[0,0,-1,0],[9E+09,9E+09,9E+09,9E+09,9E+09,9E+09]];
    CONST robtarget T4692:=[[55.750010,42.356441,48.250471],[1.000000,0.000000,0.000000,0.000000],[0,0,-1,0],[9E+09,9E+09,9E+09,9E+09,9E+09,9E+09]];
    CONST robtarget T4693:=[[55.750010,54.272228,48.250471],[1.000000,0.000000,0.000000,0.000000],[0,0,-1,0],[9E+09,9E+09,9E+09,9E+09,9E+09,9E+09]];
    CONST robtarget T4694:=[[57.250016,53.932206,48.250471],[1.000000,0.000000,0.000000,0.000000],[0,0,-1,0],[9E+09,9E+09,9E+09,9E+09,9E+09,9E+09]];
    CONST robtarget T4695:=[[57.250016,42.694188,48.250471],[1.000000,0.000000,0.000000,0.000000],[0,0,-1,0],[9E+09,9E+09,9E+09,9E+09,9E+09,9E+09]];
    CONST robtarget T4696:=[[58.750022,43.675935,48.250471],[1.000000,0.000000,0.000000,0.000000],[0,0,-1,0],[9E+09,9E+09,9E+09,9E+09,9E+09,9E+09]];
    CONST robtarget T4697:=[[58.750022,52.734294,48.250471],[1.000000,0.000000,0.000000,0.000000],[0,0,-1,0],[9E+09,9E+09,9E+09,9E+09,9E+09,9E+09]];
    CONST robtarget T4698:=[[60.250028,49.742584,48.250471],[1.000000,0.000000,0.000000,0.000000],[0,0,-1,0],[9E+09,9E+09,9E+09,9E+09,9E+09,9E+09]];
    CONST robtarget T4699:=[[60.250028,45.646615,48.250471],[1.000000,0.000000,0.000000,0.000000],[0,0,-1,0],[9E+09,9E+09,9E+09,9E+09,9E+09,9E+09]];
    CONST robtarget T4700:=[[58.750022,44.735224,48.750481],[1.000000,0.000000,0.000000,0.000000],[0,0,-1,0],[9E+09,9E+09,9E+09,9E+09,9E+09,9E+09]];
    CONST robtarget T4701:=[[58.750022,51.431005,48.750481],[1.000000,0.000000,0.000000,0.000000],[0,0,-1,0],[9E+09,9E+09,9E+09,9E+09,9E+09,9E+09]];
    CONST robtarget T4702:=[[58.750022,44.735224,48.750481],[1.000000,0.000000,0.000000,0.000000],[0,0,-1,0],[9E+09,9E+09,9E+09,9E+09,9E+09,9E+09]];
    CONST robtarget T4703:=[[58.750022,51.431005,48.750481],[1.000000,0.000000,0.000000,0.000000],[0,0,-1,0],[9E+09,9E+09,9E+09,9E+09,9E+09,9E+09]];
    CONST robtarget T4704:=[[57.250016,52.682784,48.750481],[1.000000,0.000000,0.000000,0.000000],[0,0,-1,0],[9E+09,9E+09,9E+09,9E+09,9E+09,9E+09]];
    CONST robtarget T4705:=[[57.250016,43.665420,48.750481],[1.000000,0.000000,0.000000,0.000000],[0,0,-1,0],[9E+09,9E+09,9E+09,9E+09,9E+09,9E+09]];
    CONST robtarget T4706:=[[55.750010,43.228156,48.750481],[1.000000,0.000000,0.000000,0.000000],[0,0,-1,0],[9E+09,9E+09,9E+09,9E+09,9E+09,9E+09]];
    CONST robtarget T4707:=[[55.750010,53.051624,48.750481],[1.000000,0.000000,0.000000,0.000000],[0,0,-1,0],[9E+09,9E+09,9E+09,9E+09,9E+09,9E+09]];
